   1:  PR[91,2] = PR[90,2] + -28.387;
   1:  PR[91,3] = PR[90,3] + 93.038;
   1:L PR[91] R[100]mm/sec CNT100;
   1:  PR[91,1] = PR[90,1] + 46.902;
   1:  PR[91,2] = PR[90,2] + -26.054;
   1:  PR[91,3] = PR[90,3] + 93.061;
   1:L PR[91] R[100]mm/sec CNT100;
   1:  PR[91,1] = PR[90,1] + 49.030;
   1:  PR[91,2] = PR[90,2] + -24.431;
   1:  PR[91,3] = PR[90,3] + 93.084;
   1:L PR[91] R[100]mm/sec CNT100;
   1:  PR[91,1] = PR[90,1] + 50.984;
   1:  PR[91,2] = PR[90,2] + -22.977;
   1:  PR[91,3] = PR[90,3] + 93.096;
   1:L PR[91] R[100]mm/sec CNT100;
   1:  PR[91,1] = PR[90,1] + 54.397;
   1:  PR[91,2] = PR[90,2] + -19.283;
   1:  PR[91,3] = PR[90,3] + 93.107;
   1:L PR[91] R[100]mm/sec CNT100;
   1:  PR[91,1] = PR[90,1] + 55.453;
   1:  PR[91,2] = PR[90,2] + -17.640;
   1:  PR[91,3] = PR[90,3] + 93.130;
   1:L PR[91] R[100]mm/sec CNT100;
   1:  PR[91,1] = PR[90,1] + 57.214;
   1:  PR[91,2] = PR[90,2] + -15.068;
   1:  PR[91,3] = PR[90,3] + 93.138;
   1:L PR[91] R[100]mm/sec CNT100;
   1:  PR[91,1] = PR[90,1] + 59.274;
   1:  PR[91,2] = PR[90,2] + -10.527;
   1:  PR[91,3] = PR[90,3] + 93.152;
   1:L PR[91] R[100]mm/sec CNT100;
   1:  PR[91,1] = PR[90,1] + 60.517;
   1:  PR[91,2] = PR[90,2] + -5.701;
   1:  PR[91,3] = PR[90,3] + 93.174;
   1:L PR[91] R[100]mm/sec CNT100;
   1:  PR[91,1] = PR[90,1] + 60.793;
   1:  PR[91,2] = PR[90,2] + -2.425;
   1:  PR[91,3] = PR[90,3] + 93.197;
   1:L PR[91] R[100]mm/sec CNT100;
   1:  PR[91,1] = PR[90,1] + 60.883;
   1:  PR[91,2] = PR[90,2] + -0.761;
   1:  PR[91,3] = PR[90,3] + 93.211;
   1:L PR[91] R[100]mm/sec CNT100;
   1:  PR[91,1] = PR[90,1] + 60.748;
   1:  PR[91,2] = PR[90,2] + 0.799;
   1:  PR[91,3] = PR[90,3] + 93.219;
   1:L PR[91] R[100]mm/sec CNT100;
   1:  PR[91,1] = PR[90,1] + 60.667;
   1:  PR[91,2] = PR[90,2] + 2.423;
   1:  PR[91,3] = PR[90,3] + 93.226;
   1:L PR[91] R[100]mm/sec CNT100;
   1:  PR[91,1] = PR[90,1] + 60.517;
   1:  PR[91,2] = PR[90,2] + 4.243;
   1:  PR[91,3] = PR[90,3] + 93.233;
   1:L PR[91] R[100]mm/sec CNT100;
   1:  PR[91,1] = PR[90,1] + 59.274;
   1:  PR[91,2] = PR[90,2] + 9.068;
   1:  PR[91,3] = PR[90,3] + 93.241;
   1:L PR[91] R[100]mm/sec CNT100;
   1:  PR[91,1] = PR[90,1] + 57.214;
   1:  PR[91,2] = PR[90,2] + 13.609;
   1:  PR[91,3] = PR[90,3] + 93.263;
   1:L PR[91] R[100]mm/sec CNT100;
   1:  PR[91,1] = PR[90,1] + 55.453;
   1:  PR[91,2] = PR[90,2] + 16.181;
   1:  PR[91,3] = PR[90,3] + 93.285;
   1:L PR[91] R[100]mm/sec CNT100;
   1:  PR[91,1] = PR[90,1] + 54.397;
   1:  PR[91,2] = PR[90,2] + 17.825;
   1:  PR[91,3] = PR[90,3] + 93.299;
   1:L PR[91] R[100]mm/sec CNT100;
   1:  PR[91,1] = PR[90,1] + 50.984;
   1:  PR[91,2] = PR[90,2] + 21.518;
   1:  PR[91,3] = PR[90,3] + 93.308;
   1:L PR[91] R[100]mm/sec CNT100;
   1:  PR[91,1] = PR[90,1] + 49.030;
   1:  PR[91,2] = PR[90,2] + 22.972;
   1:  PR[91,3] = PR[90,3] + 93.330;
   1:L PR[91] R[100]mm/sec CNT100;
   1:  PR[91,1] = PR[90,1] + 46.902;
   1:  PR[91,2] = PR[90,2] + 24.595;
   1:  PR[91,3] = PR[90,3] + 93.341;
   1:L PR[91] R[100]mm/sec CNT100;
   1:  PR[91,1] = PR[90,1] + 42.292;
   1:  PR[91,2] = PR[90,2] + 26.928;
   1:  PR[91,3] = PR[90,3] + 93.353;
   1:L PR[91] R[100]mm/sec CNT100;
   1:  PR[91,1] = PR[90,1] + 37.245;
   1:  PR[91,2] = PR[90,2] + 28.447;
   1:  PR[91,3] = PR[90,3] + 93.376;
   1:L PR[91] R[100]mm/sec CNT100;
   1:  PR[91,1] = PR[90,1] + 32.511;
   1:  PR[91,2] = PR[90,2] + 29.043;
   1:  PR[91,3] = PR[90,3] + 93.399;
   1:L PR[91] R[100]mm/sec CNT100;
   1:  PR[91,1] = PR[90,1] + 31.765;
   1:  PR[91,2] = PR[90,2] + 29.058;
   1:  PR[91,3] = PR[90,3] + 93.421;
   1:L PR[91] R[100]mm/sec CNT100;
   1:  PR[91,1] = PR[90,1] + 27.568;
   1:  PR[91,2] = PR[90,2] + 28.827;
   1:  PR[91,3] = PR[90,3] + 93.424;
   1:L PR[91] R[100]mm/sec CNT100;
   1:  PR[91,1] = PR[90,1] + 26.159;
   1:  PR[91,2] = PR[90,2] + 28.598;
   1:  PR[91,3] = PR[90,3] + 93.443;
   1:L PR[91] R[100]mm/sec CNT100;
   1:  PR[91,1] = PR[90,1] + 21.407;
   1:  PR[91,2] = PR[90,2] + 27.464;
   1:  PR[91,3] = PR[90,3] + 93.449;
   1:L PR[91] R[100]mm/sec CNT100;
   1:  PR[91,1] = PR[90,1] + 20.575;
   1:  PR[91,2] = PR[90,2] + 27.472;
   1:  PR[91,3] = PR[90,3] + 93.471;
   1:L PR[91] R[100]mm/sec CNT100;
   1:  PR[91,1] = PR[90,1] + 19.235;
   1:  PR[91,2] = PR[90,2] + 27.410;
   1:  PR[91,3] = PR[90,3] + 93.474;
   1:L PR[91] R[100]mm/sec CNT100;
   1:  PR[91,1] = PR[90,1] + 18.275;
   1:  PR[91,2] = PR[90,2] + 27.467;
   1:  PR[91,3] = PR[90,3] + 93.480;
   1:L PR[91] R[100]mm/sec CNT100;
   1:  PR[91,1] = PR[90,1] + 7.525;
   1:  PR[91,2] = PR[90,2] + 27.884;
   1:  PR[91,3] = PR[90,3] + 93.485;
   1:L PR[91] R[100]mm/sec CNT100;
   1:  PR[91,1] = PR[90,1] + -2.993;
   1:  PR[91,2] = PR[90,2] + 27.478;
   1:  PR[91,3] = PR[90,3] + 93.533;
   1:L PR[91] R[100]mm/sec CNT100;
   1:  PR[91,1] = PR[90,1] + -5.796;
   1:  PR[91,2] = PR[90,2] + 27.186;
   1:  PR[91,3] = PR[90,3] + 93.579;
   1:L PR[91] R[100]mm/sec CNT100;
   1:  PR[91,1] = PR[90,1] + -13.027;
   1:  PR[91,2] = PR[90,2] + 26.396;
   1:  PR[91,3] = PR[90,3] + 93.592;
   1:L PR[91] R[100]mm/sec CNT100;
   1:  PR[91,1] = PR[90,1] + -18.279;
   1:  PR[91,2] = PR[90,2] + 25.461;
   1:  PR[91,3] = PR[90,3] + 93.624;
   1:L PR[91] R[100]mm/sec CNT100;
   1:  PR[91,1] = PR[90,1] + -22.384;
   1:  PR[91,2] = PR[90,2] + 24.710;
   1:  PR[91,3] = PR[90,3] + 93.648;
   1:L PR[91] R[100]mm/sec CNT100;
   1:  PR[91,1] = PR[90,1] + -30.899;
   1:  PR[91,2] = PR[90,2] + 22.489;
   1:  PR[91,3] = PR[90,3] + 93.667;
   1:L PR[91] R[100]mm/sec CNT100;
   1:  PR[91,1] = PR[90,1] + -36.804;
   1:  PR[91,2] = PR[90,2] + 20.391;
   1:  PR[91,3] = PR[90,3] + 93.706;
   1:L PR[91] R[100]mm/sec CNT100;
   1:  PR[91,1] = PR[90,1] + -37.835;
   1:  PR[91,2] = PR[90,2] + 19.997;
   1:  PR[91,3] = PR[90,3] + 93.734;
   1:L PR[91] R[100]mm/sec CNT100;
   1:  PR[91,1] = PR[90,1] + -38.951;
   1:  PR[91,2] = PR[90,2] + 19.482;
   1:  PR[91,3] = PR[90,3] + 93.739;
   1:L PR[91] R[100]mm/sec CNT100;
   1:  PR[91,1] = PR[90,1] + -43.041;
   1:  PR[91,2] = PR[90,2] + 17.397;
   1:  PR[91,3] = PR[90,3] + 93.744;
   1:L PR[91] R[100]mm/sec CNT100;
   1:  PR[91,1] = PR[90,1] + -48.727;
   1:  PR[91,2] = PR[90,2] + 13.596;
   1:  PR[91,3] = PR[90,3] + 93.765;
   1:L PR[91] R[100]mm/sec CNT100;
   1:  PR[91] = PR[90];
   1:  PR[91,1] = PR[90,1] + -49.365;
   1:  PR[91,2] = PR[90,2] + 11.172;
   1:  PR[91,3] = PR[90,3] + 95.095;
   1:L PR[91] R[100]mm/sec CNT100;
   1:  PR[91,1] = PR[90,1] + -51.153;
   1:  PR[91,2] = PR[90,2] + 9.107;
   1:  PR[91,3] = PR[90,3] + 93.811;
   1:L PR[91] R[100]mm/sec CNT100;
   1:  PR[91,1] = PR[90,1] + -51.534;
   1:  PR[91,2] = PR[90,2] + 8.367;
   1:  PR[91,3] = PR[90,3] + 93.823;
   1:L PR[91] R[100]mm/sec CNT100;
   1:  PR[91,1] = PR[90,1] + -53.546;
   1:  PR[91,2] = PR[90,2] + 4.268;
   1:  PR[91,3] = PR[90,3] + 93.827;
   1:L PR[91] R[100]mm/sec CNT100;
   1:  PR[91,1] = PR[90,1] + -53.848;
   1:  PR[91,2] = PR[90,2] + 2.477;
   1:  PR[91,3] = PR[90,3] + 93.847;
   1:L PR[91] R[100]mm/sec CNT100;
   1:  PR[91,1] = PR[90,1] + -54.520;
   1:  PR[91,2] = PR[90,2] + -0.745;
   1:  PR[91,3] = PR[90,3] + 93.856;
   1:L PR[91] R[100]mm/sec CNT100;
   1:  PR[91,1] = PR[90,1] + -54.513;
   1:  PR[91,2] = PR[90,2] + -0.783;
   1:  PR[91,3] = PR[90,3] + 93.870;
   1:L PR[91] R[100]mm/sec CNT100;
   1:  PR[91,1] = PR[90,1] + -54.240;
   1:  PR[91,2] = PR[90,2] + -1.528;
   1:  PR[91,3] = PR[90,3] + 93.871;
   1:L PR[91] R[100]mm/sec CNT100;
   1:  PR[91,1] = PR[90,1] + -53.592;
   1:  PR[91,2] = PR[90,2] + -5.660;
   1:  PR[91,3] = PR[90,3] + 93.874;
   1:L PR[91] R[100]mm/sec CNT100;
   1:  PR[91,1] = PR[90,1] + -53.290;
   1:  PR[91,2] = PR[90,2] + -6.306;
   1:  PR[91,3] = PR[90,3] + 93.893;
   1:L PR[91] R[100]mm/sec CNT100;
   1:  PR[91,1] = PR[90,1] + -51.237;
   1:  PR[91,2] = PR[90,2] + -10.564;
   1:  PR[91,3] = PR[90,3] + 93.896;
   1:L PR[91] R[100]mm/sec CNT100;
   1:  PR[91,1] = PR[90,1] + -50.866;
   1:  PR[91,2] = PR[90,2] + -11.004;
   1:  PR[91,3] = PR[90,3] + 93.917;
   1:L PR[91] R[100]mm/sec CNT100;
   1:  PR[91,1] = PR[90,1] + -47.495;
   1:  PR[91,2] = PR[90,2] + -14.421;
   1:  PR[91,3] = PR[90,3] + 93.920;
   1:L PR[91] R[100]mm/sec CNT100;
   1:  PR[91,1] = PR[90,1] + -46.719;
   1:  PR[91,2] = PR[90,2] + -15.165;
   1:  PR[91,3] = PR[90,3] + 93.942;
   1:L PR[91] R[100]mm/sec CNT100;
   1:  PR[91,1] = PR[90,1] + -44.576;
   1:  PR[91,2] = PR[90,2] + -16.660;
   1:  PR[91,3] = PR[90,3] + 93.946;
   1:L PR[91] R[100]mm/sec CNT100;
   1:  PR[91,1] = PR[90,1] + -41.398;
   1:  PR[91,2] = PR[90,2] + -18.787;
   1:  PR[91,3] = PR[90,3] + 93.958;
   1:L PR[91] R[100]mm/sec CNT100;
   1:  PR[91,1] = PR[90,1] + -37.258;
   1:  PR[91,2] = PR[90,2] + -20.921;
   1:  PR[91,3] = PR[90,3] + 93.975;
   1:L PR[91] R[100]mm/sec CNT100;
   1:  PR[91,1] = PR[90,1] + -36.150;
   1:  PR[91,2] = PR[90,2] + -21.445;
   1:  PR[91,3] = PR[90,3] + 93.996;
   1:L PR[91] R[100]mm/sec CNT100;
   1:  PR[91,1] = PR[90,1] + -28.560;
   1:  PR[91,2] = PR[90,2] + -24.144;
   1:  PR[91,3] = PR[90,3] + 94.002;
   1:L PR[91] R[100]mm/sec CNT100;
   1:  PR[91,1] = PR[90,1] + -19.983;
   1:  PR[91,2] = PR[90,2] + -26.385;
   1:  PR[91,3] = PR[90,3] + 94.038;
   1:L PR[91] R[100]mm/sec CNT100;
   1:  PR[91,1] = PR[90,1] + -15.009;
   1:  PR[91,2] = PR[90,2] + -27.294;
   1:  PR[91,3] = PR[90,3] + 94.078;
   1:L PR[91] R[100]mm/sec CNT100;
   1:  PR[91,1] = PR[90,1] + -10.557;
   1:  PR[91,2] = PR[90,2] + -28.087;
   1:  PR[91,3] = PR[90,3] + 94.101;
   1:L PR[91] R[100]mm/sec CNT100;
   1:  PR[91,1] = PR[90,1] + -0.444;
   1:  PR[91,2] = PR[90,2] + -29.181;
   1:  PR[91,3] = PR[90,3] + 94.121;
   1:L PR[91] R[100]mm/sec CNT100;
   1:  PR[91,1] = PR[90,1] + 6.896;
   1:  PR[91,2] = PR[90,2] + -29.464;
   1:  PR[91,3] = PR[90,3] + 94.167;
   1:L PR[91] R[100]mm/sec CNT100;
   1:  PR[91,1] = PR[90,1] + 9.665;
   1:  PR[91,2] = PR[90,2] + -29.600;
   1:  PR[91,3] = PR[90,3] + 94.200;
   1:L PR[91] R[100]mm/sec CNT100;
   1:  PR[91,1] = PR[90,1] + 13.880;
   1:  PR[91,2] = PR[90,2] + -29.451;
   1:  PR[91,3] = PR[90,3] + 94.212;
   1:L PR[91] R[100]mm/sec CNT100;
   1:  PR[91,1] = PR[90,1] + 21.353;
   1:  PR[91,2] = PR[90,2] + -29.130;
   1:  PR[91,3] = PR[90,3] + 94.231;
   1:L PR[91] R[100]mm/sec CNT100;
   1:  PR[91,1] = PR[90,1] + 25.563;
   1:  PR[91,2] = PR[90,2] + -30.127;
   1:  PR[91,3] = PR[90,3] + 94.265;
   1:L PR[91] R[100]mm/sec CNT100;
   1:  PR[91,1] = PR[90,1] + 27.869;
   1:  PR[91,2] = PR[90,2] + -30.501;
   1:  PR[91,3] = PR[90,3] + 94.284;
   1:L PR[91] R[100]mm/sec CNT100;
   1:  PR[91,1] = PR[90,1] + 31.160;
   1:  PR[91,2] = PR[90,2] + -30.682;
   1:  PR[91,3] = PR[90,3] + 94.295;
   1:L PR[91] R[100]mm/sec CNT100;
   1:  PR[91,1] = PR[90,1] + 32.947;
   1:  PR[91,2] = PR[90,2] + -30.648;
   1:  PR[91,3] = PR[90,3] + 94.310;
   1:L PR[91] R[100]mm/sec CNT100;
   1:  PR[91,1] = PR[90,1] + 36.769;
   1:  PR[91,2] = PR[90,2] + -30.166;
   1:  PR[91,3] = PR[90,3] + 94.318;
   1:L PR[91] R[100]mm/sec CNT100;
   1:  PR[91,1] = PR[90,1] + 37.799;
   1:  PR[91,2] = PR[90,2] + -29.954;
   1:  PR[91,3] = PR[90,3] + 94.335;
   1:L PR[91] R[100]mm/sec CNT100;
   1:  PR[91,1] = PR[90,1] + 42.128;
   1:  PR[91,2] = PR[90,2] + -28.597;
   1:  PR[91,3] = PR[90,3] + 94.340;
   1:L PR[91] R[100]mm/sec CNT100;
   1:  PR[91,1] = PR[90,1] + 42.265;
   1:  PR[91,2] = PR[90,2] + -28.541;
   1:  PR[91,3] = PR[90,3] + 94.360;
   1:L PR[91] R[100]mm/sec CNT100;
   1:  PR[91,1] = PR[90,1] + 43.627;
   1:  PR[91,2] = PR[90,2] + -27.829;
   1:  PR[91,3] = PR[90,3] + 94.361;
   1:L PR[91] R[100]mm/sec CNT100;
   1:  PR[91,1] = PR[90,1] + 46.813;
   1:  PR[91,2] = PR[90,2] + -26.224;
   1:  PR[91,3] = PR[90,3] + 94.368;
   1:L PR[91] R[100]mm/sec CNT100;
   1:  PR[91,1] = PR[90,1] + 50.933;
   1:  PR[91,2] = PR[90,2] + -23.145;
   1:  PR[91,3] = PR[90,3] + 94.384;
   1:L PR[91] R[100]mm/sec CNT100;
   1:  PR[91,1] = PR[90,1] + 52.529;
   1:  PR[91,2] = PR[90,2] + -21.411;
   1:  PR[91,3] = PR[90,3] + 94.407;
   1:L PR[91] R[100]mm/sec CNT100;
   1:  PR[91,1] = PR[90,1] + 54.411;
   1:  PR[91,2] = PR[90,2] + -19.423;
   1:  PR[91,3] = PR[90,3] + 94.418;
   1:L PR[91] R[100]mm/sec CNT100;
   1:  PR[91,1] = PR[90,1] + 56.574;
   1:  PR[91,2] = PR[90,2] + -16.056;
   1:  PR[91,3] = PR[90,3] + 94.430;
   1:L PR[91] R[100]mm/sec CNT100;
   1:  PR[91,1] = PR[90,1] + 57.151;
   1:  PR[91,2] = PR[90,2] + -15.186;
   1:  PR[91,3] = PR[90,3] + 94.448;
   1:L PR[91] R[100]mm/sec CNT100;
   1:  PR[91,1] = PR[90,1] + 58.813;
   1:  PR[91,2] = PR[90,2] + -11.280;
   1:  PR[91,3] = PR[90,3] + 94.453;
   1:L PR[91] R[100]mm/sec CNT100;
   1:  PR[91,1] = PR[90,1] + 59.145;
   1:  PR[91,2] = PR[90,2] + -10.551;
   1:  PR[91,3] = PR[90,3] + 94.472;
   1:L PR[91] R[100]mm/sec CNT100;
   1:  PR[91,1] = PR[90,1] + 60.403;
   1:  PR[91,2] = PR[90,2] + -5.711;
   1:  PR[91,3] = PR[90,3] + 94.475;
   1:L PR[91] R[100]mm/sec CNT100;
   1:  PR[91,1] = PR[90,1] + 60.481;
   1:  PR[91,2] = PR[90,2] + -4.788;
   1:  PR[91,3] = PR[90,3] + 94.498;
   1:L PR[91] R[100]mm/sec CNT100;
   1:  PR[91,1] = PR[90,1] + 60.550;
   1:  PR[91,2] = PR[90,2] + -3.505;
   1:  PR[91,3] = PR[90,3] + 94.502;
   1:L PR[91] R[100]mm/sec CNT100;
   1:  PR[91,1] = PR[90,1] + 60.782;
   1:  PR[91,2] = PR[90,2] + -0.697;
   1:  PR[91,3] = PR[90,3] + 94.508;
   1:L PR[91] R[100]mm/sec CNT100;
   1:  PR[91,1] = PR[90,1] + 60.735;
   1:  PR[91,2] = PR[90,2] + 0.247;
   1:  PR[91,3] = PR[90,3] + 94.521;
   1:L PR[91] R[100]mm/sec CNT100;
   1:  PR[91,1] = PR[90,1] + 60.403;
   1:  PR[91,2] = PR[90,2] + 4.253;
   1:  PR[91,3] = PR[90,3] + 94.525;
   1:L PR[91] R[100]mm/sec CNT100;
   1:  PR[91,1] = PR[90,1] + 59.145;
   1:  PR[91,2] = PR[90,2] + 9.092;
   1:  PR[91,3] = PR[90,3] + 94.543;
   1:L PR[91] R[100]mm/sec CNT100;
   1:  PR[91,1] = PR[90,1] + 58.813;
   1:  PR[91,2] = PR[90,2] + 9.821;
   1:  PR[91,3] = PR[90,3] + 94.565;
   1:L PR[91] R[100]mm/sec CNT100;
   1:  PR[91,1] = PR[90,1] + 57.151;
   1:  PR[91,2] = PR[90,2] + 13.728;
   1:  PR[91,3] = PR[90,3] + 94.569;
   1:L PR[91] R[100]mm/sec CNT100;
   1:  PR[91,1] = PR[90,1] + 56.574;
   1:  PR[91,2] = PR[90,2] + 14.597;
   1:  PR[91,3] = PR[90,3] + 94.588;
   1:L PR[91] R[100]mm/sec CNT100;
   1:  PR[91,1] = PR[90,1] + 54.411;
   1:  PR[91,2] = PR[90,2] + 17.964;
   1:  PR[91,3] = PR[90,3] + 94.593;
   1:L PR[91] R[100]mm/sec CNT100;
   1:  PR[91,1] = PR[90,1] + 52.529;
   1:  PR[91,2] = PR[90,2] + 19.953;
   1:  PR[91,3] = PR[90,3] + 94.611;
   1:L PR[91] R[100]mm/sec CNT100;
   1:  PR[91,1] = PR[90,1] + 50.933;
   1:  PR[91,2] = PR[90,2] + 21.686;
   1:  PR[91,3] = PR[90,3] + 94.623;
   1:L PR[91] R[100]mm/sec CNT100;
   1:  PR[91,1] = PR[90,1] + 46.813;
   1:  PR[91,2] = PR[90,2] + 24.766;
   1:  PR[91,3] = PR[90,3] + 94.634;
   1:L PR[91] R[100]mm/sec CNT100;
   1:  PR[91,1] = PR[90,1] + 43.627;
   1:  PR[91,2] = PR[90,2] + 26.370;
   1:  PR[91,3] = PR[90,3] + 94.657;
   1:L PR[91] R[100]mm/sec CNT100;
   1:  PR[91,1] = PR[90,1] + 42.266;
   1:  PR[91,2] = PR[90,2] + 27.082;
   1:  PR[91,3] = PR[90,3] + 94.673;
   1:L PR[91] R[100]mm/sec CNT100;
   1:  PR[91,1] = PR[90,1] + 42.128;
   1:  PR[91,2] = PR[90,2] + 27.139;
   1:  PR[91,3] = PR[90,3] + 94.680;
   1:L PR[91] R[100]mm/sec CNT100;
   1:  PR[91,1] = PR[90,1] + 37.800;
   1:  PR[91,2] = PR[90,2] + 28.494;
   1:L PR[91] R[100]mm/sec CNT100;
   1:  PR[91,1] = PR[90,1] + 36.772;
   1:  PR[91,2] = PR[90,2] + 28.707;
   1:  PR[91,3] = PR[90,3] + 94.701;
   1:L PR[91] R[100]mm/sec CNT100;
   1:  PR[91,1] = PR[90,1] + 32.950;
   1:  PR[91,2] = PR[90,2] + 29.189;
   1:  PR[91,3] = PR[90,3] + 94.706;
   1:L PR[91] R[100]mm/sec CNT100;
   1:  PR[91,1] = PR[90,1] + 31.164;
   1:  PR[91,2] = PR[90,2] + 29.224;
   1:  PR[91,3] = PR[90,3] + 94.723;
   1:L PR[91] R[100]mm/sec CNT100;
   1:  PR[91,1] = PR[90,1] + 27.875;
   1:  PR[91,2] = PR[90,2] + 29.043;
   1:  PR[91,3] = PR[90,3] + 94.731;
   1:L PR[91] R[100]mm/sec CNT100;
   1:  PR[91,1] = PR[90,1] + 25.550;
   1:  PR[91,2] = PR[90,2] + 28.666;
   1:  PR[91,3] = PR[90,3] + 94.746;
   1:L PR[91] R[100]mm/sec CNT100;
   1:  PR[91,1] = PR[90,1] + 21.358;
   1:  PR[91,2] = PR[90,2] + 27.673;
   1:  PR[91,3] = PR[90,3] + 94.756;
   1:L PR[91] R[100]mm/sec CNT100;
   1:  PR[91,1] = PR[90,1] + 9.661;
   1:  PR[91,2] = PR[90,2] + 28.141;
   1:  PR[91,3] = PR[90,3] + 94.776;
   1:L PR[91] R[100]mm/sec CNT100;
   1:  PR[91,1] = PR[90,1] + 6.896;
   1:  PR[91,2] = PR[90,2] + 28.005;
   1:  PR[91,3] = PR[90,3] + 94.828;
   1:L PR[91] R[100]mm/sec CNT100;
   1:  PR[91,1] = PR[90,1] + -0.444;
   1:  PR[91,2] = PR[90,2] + 27.723;
   1:  PR[91,3] = PR[90,3] + 94.841;
   1:L PR[91] R[100]mm/sec CNT100;
   1:  PR[91,1] = PR[90,1] + -10.557;
   1:  PR[91,2] = PR[90,2] + 26.628;
   1:  PR[91,3] = PR[90,3] + 94.874;
   1:L PR[91] R[100]mm/sec CNT100;
   1:  PR[91,1] = PR[90,1] + -15.009;
   1:  PR[91,2] = PR[90,2] + 25.835;
   1:  PR[91,3] = PR[90,3] + 94.920;
   1:L PR[91] R[100]mm/sec CNT100;
   1:  PR[91,1] = PR[90,1] + -19.983;
   1:  PR[91,2] = PR[90,2] + 24.926;
   1:  PR[91,3] = PR[90,3] + 94.940;
   1:L PR[91] R[100]mm/sec CNT100;
   1:  PR[91,1] = PR[90,1] + -28.560;
   1:  PR[91,2] = PR[90,2] + 22.685;
   1:  PR[91,3] = PR[90,3] + 94.963;
   1:L PR[91] R[100]mm/sec CNT100;
   1:  PR[91,1] = PR[90,1] + -36.150;
   1:  PR[91,2] = PR[90,2] + 19.987;
   1:  PR[91,3] = PR[90,3] + 95.003;
   1:L PR[91] R[100]mm/sec CNT100;
   1:  PR[91,1] = PR[90,1] + -37.263;
   1:  PR[91,2] = PR[90,2] + 19.461;
   1:  PR[91,3] = PR[90,3] + 95.039;
   1:L PR[91] R[100]mm/sec CNT100;
   1:  PR[91,1] = PR[90,1] + -41.425;
   1:  PR[91,2] = PR[90,2] + 17.338;
   1:  PR[91,3] = PR[90,3] + 95.044;
   1:L PR[91] R[100]mm/sec CNT100;
   1:  PR[91,1] = PR[90,1] + -45.308;
   1:  PR[91,2] = PR[90,2] + 14.742;
   1:  PR[91,3] = PR[90,3] + 95.065;
   1:L PR[91] R[100]mm/sec CNT100;
   1:  PR[91,1] = PR[90,1] + -46.871;
   1:  PR[91,2] = PR[90,2] + 13.661;
   1:  PR[91,3] = PR[90,3] + 95.086;
   1:L PR[91] R[100]mm/sec CNT100;
   1:  PR[91] = PR[90];
   1:  PR[91,1] = PR[90,1] + -49.712;
   1:  PR[91,2] = PR[90,2] + 9.014;
   1:  PR[91,3] = PR[90,3] + 96.395;
   1:L PR[91] R[100]mm/sec CNT100;
   1:  PR[91,1] = PR[90,1] + -49.895;
   1:  PR[91,2] = PR[90,2] + 8.687;
   1:  PR[91,3] = PR[90,3] + 95.126;
   1:L PR[91] R[100]mm/sec CNT100;
   1:  PR[91,1] = PR[90,1] + -52.067;
   1:  PR[91,2] = PR[90,2] + 4.259;
   1:  PR[91,3] = PR[90,3] + 95.127;
   1:L PR[91] R[100]mm/sec CNT100;
   1:  PR[91,1] = PR[90,1] + -52.198;
   1:  PR[91,2] = PR[90,2] + 3.486;
   1:  PR[91,3] = PR[90,3] + 95.150;
   1:L PR[91] R[100]mm/sec CNT100;
   1:  PR[91,1] = PR[90,1] + -52.873;
   1:  PR[91,2] = PR[90,2] + 0.250;
   1:  PR[91,3] = PR[90,3] + 95.153;
   1:L PR[91] R[100]mm/sec CNT100;
   1:  PR[91,1] = PR[90,1] + -53.010;
   1:  PR[91,2] = PR[90,2] + -0.543;
   1:  PR[91,3] = PR[90,3] + 95.168;
   1:L PR[91] R[100]mm/sec CNT100;
   1:  PR[91,1] = PR[90,1] + -52.918;
   1:  PR[91,2] = PR[90,2] + -0.793;
   1:  PR[91,3] = PR[90,3] + 95.172;
   1:L PR[91] R[100]mm/sec CNT100;
   1:  PR[91,1] = PR[90,1] + -52.146;
   1:  PR[91,2] = PR[90,2] + -5.720;
   1:  PR[91,3] = PR[90,3] + 95.173;
   1:L PR[91] R[100]mm/sec CNT100;
   1:  PR[91,1] = PR[90,1] + -51.429;
   1:  PR[91,2] = PR[90,2] + -7.208;
   1:  PR[91,3] = PR[90,3] + 95.196;
   1:L PR[91] R[100]mm/sec CNT100;
   1:  PR[91,1] = PR[90,1] + -49.680;
   1:  PR[91,2] = PR[90,2] + -10.338;
   1:  PR[91,3] = PR[90,3] + 95.203;
   1:L PR[91] R[100]mm/sec CNT100;
   1:  PR[91,1] = PR[90,1] + -49.463;
   1:  PR[91,2] = PR[90,2] + -10.639;
   1:  PR[91,3] = PR[90,3] + 95.219;
   1:L PR[91] R[100]mm/sec CNT100;
   1:  PR[91,1] = PR[90,1] + -46.177;
   1:  PR[91,2] = PR[90,2] + -13.970;
   1:  PR[91,3] = PR[90,3] + 95.221;
   1:L PR[91] R[100]mm/sec CNT100;
   1:  PR[91,1] = PR[90,1] + -44.827;
   1:  PR[91,2] = PR[90,2] + -15.265;
   1:  PR[91,3] = PR[90,3] + 95.242;
   1:L PR[91] R[100]mm/sec CNT100;
   1:  PR[91,1] = PR[90,1] + -41.238;
   1:  PR[91,2] = PR[90,2] + -17.768;
   1:  PR[91,3] = PR[90,3] + 95.251;
   1:L PR[91] R[100]mm/sec CNT100;
   1:  PR[91,1] = PR[90,1] + -39.794;
   1:  PR[91,2] = PR[90,2] + -18.734;
   1:  PR[91,3] = PR[90,3] + 95.270;
   1:L PR[91] R[100]mm/sec CNT100;
   1:  PR[91,1] = PR[90,1] + -37.907;
   1:  PR[91,2] = PR[90,2] + -19.708;
   1:  PR[91,3] = PR[90,3] + 95.278;
   1:L PR[91] R[100]mm/sec CNT100;
   1:  PR[91,1] = PR[90,1] + -33.865;
   1:  PR[91,2] = PR[90,2] + -21.618;
   1:  PR[91,3] = PR[90,3] + 95.288;
   1:L PR[91] R[100]mm/sec CNT100;
   1:  PR[91,1] = PR[90,1] + -26.220;
   1:  PR[91,2] = PR[90,2] + -24.340;
   1:  PR[91,3] = PR[90,3] + 95.308;
   1:L PR[91] R[100]mm/sec CNT100;
   1:  PR[91,1] = PR[90,1] + -17.581;
   1:  PR[91,2] = PR[90,2] + -26.600;
   1:  PR[91,3] = PR[90,3] + 95.345;
   1:L PR[91] R[100]mm/sec CNT100;
   1:  PR[91,1] = PR[90,1] + -11.739;
   1:  PR[91,2] = PR[90,2] + -27.669;
   1:  PR[91,3] = PR[90,3] + 95.385;
   1:L PR[91] R[100]mm/sec CNT100;
   1:  PR[91,1] = PR[90,1] + -8.086;
   1:  PR[91,2] = PR[90,2] + -28.319;
   1:  PR[91,3] = PR[90,3] + 95.412;
   1:L PR[91] R[100]mm/sec CNT100;
   1:  PR[91,1] = PR[90,1] + 1.029;
   1:  PR[91,2] = PR[90,2] + -29.314;
   1:  PR[91,3] = PR[90,3] + 95.429;
   1:L PR[91] R[100]mm/sec CNT100;
   1:  PR[91,1] = PR[90,1] + 2.098;
   1:  PR[91,2] = PR[90,2] + -29.426;
   1:  PR[91,3] = PR[90,3] + 95.471;
   1:L PR[91] R[100]mm/sec CNT100;
   1:  PR[91,1] = PR[90,1] + 6.247;
   1:  PR[91,2] = PR[90,2] + -29.586;
   1:  PR[91,3] = PR[90,3] + 95.475;
   1:L PR[91] R[100]mm/sec CNT100;
   1:  PR[91,1] = PR[90,1] + 11.792;
   1:  PR[91,2] = PR[90,2] + -29.857;
   1:  PR[91,3] = PR[90,3] + 95.494;
   1:L PR[91] R[100]mm/sec CNT100;
   1:  PR[91,1] = PR[90,1] + 14.899;
   1:  PR[91,2] = PR[90,2] + -29.747;
   1:  PR[91,3] = PR[90,3] + 95.519;
   1:L PR[91] R[100]mm/sec CNT100;
   1:  PR[91,1] = PR[90,1] + 20.303;
   1:  PR[91,2] = PR[90,2] + -29.520;
   1:  PR[91,3] = PR[90,3] + 95.533;
   1:L PR[91] R[100]mm/sec CNT100;
   1:  PR[91,1] = PR[90,1] + 24.444;
   1:  PR[91,2] = PR[90,2] + -29.300;
   1:  PR[91,3] = PR[90,3] + 95.558;
   1:L PR[91] R[100]mm/sec CNT100;
   1:  PR[91,1] = PR[90,1] + 24.240;
   1:  PR[91,2] = PR[90,2] + -30.026;
   1:  PR[91,3] = PR[90,3] + 95.577;
   1:L PR[91] R[100]mm/sec CNT100;
   1:  PR[91,1] = PR[90,1] + 24.959;
   1:  PR[91,2] = PR[90,2] + -30.195;
   1:  PR[91,3] = PR[90,3] + 95.580;
   1:L PR[91] R[100]mm/sec CNT100;
   1:  PR[91,1] = PR[90,1] + 28.174;
   1:  PR[91,2] = PR[90,2] + -30.717;
   1:  PR[91,3] = PR[90,3] + 95.583;
   1:L PR[91] R[100]mm/sec CNT100;
   1:  PR[91,1] = PR[90,1] + 30.556;
   1:  PR[91,2] = PR[90,2] + -30.848;
   1:  PR[91,3] = PR[90,3] + 95.598;
   1:L PR[91] R[100]mm/sec CNT100;
   1:  PR[91,1] = PR[90,1] + 33.384;
   1:  PR[91,2] = PR[90,2] + -30.793;
   1:  PR[91,3] = PR[90,3] + 95.609;
   1:L PR[91] R[100]mm/sec CNT100;
   1:  PR[91,1] = PR[90,1] + 36.206;
   1:  PR[91,2] = PR[90,2] + -30.438;
   1:  PR[91,3] = PR[90,3] + 95.622;
   1:L PR[91] R[100]mm/sec CNT100;
   1:  PR[91,1] = PR[90,1] + 38.380;
   1:  PR[91,2] = PR[90,2] + -29.988;
   1:  PR[91,3] = PR[90,3] + 95.635;
   1:L PR[91] R[100]mm/sec CNT100;
   1:  PR[91,1] = PR[90,1] + 41.632;
   1:  PR[91,2] = PR[90,2] + -28.969;
   1:  PR[91,3] = PR[90,3] + 95.645;
   1:L PR[91] R[100]mm/sec CNT100;
   1:  PR[91,1] = PR[90,1] + 42.997;
   1:  PR[91,2] = PR[90,2] + -28.411;
   1:  PR[91,3] = PR[90,3] + 95.660;
   1:L PR[91] R[100]mm/sec CNT100;
   1:  PR[91,1] = PR[90,1] + 46.615;
   1:  PR[91,2] = PR[90,2] + -26.519;
   1:  PR[91,3] = PR[90,3] + 95.667;
   1:L PR[91] R[100]mm/sec CNT100;
   1:  PR[91,1] = PR[90,1] + 47.102;
   1:  PR[91,2] = PR[90,2] + -26.205;
   1:  PR[91,3] = PR[90,3] + 95.685;
   1:L PR[91] R[100]mm/sec CNT100;
   1:  PR[91,1] = PR[90,1] + 49.866;
   1:  PR[91,2] = PR[90,2] + -24.067;
   1:  PR[91,3] = PR[90,3] + 95.688;
   1:L PR[91] R[100]mm/sec CNT100;
   1:  PR[91,1] = PR[90,1] + 50.896;
   1:  PR[91,2] = PR[90,2] + -23.301;
   1:  PR[91,3] = PR[90,3] + 95.704;
   1:L PR[91] R[100]mm/sec CNT100;
   1:  PR[91,1] = PR[90,1] + 54.418;
   1:  PR[91,2] = PR[90,2] + -19.573;
   1:  PR[91,3] = PR[90,3] + 95.710;
   1:L PR[91] R[100]mm/sec CNT100;
   1:  PR[91,1] = PR[90,1] + 55.294;
   1:  PR[91,2] = PR[90,2] + -18.209;
   1:  PR[91,3] = PR[90,3] + 95.733;
   1:L PR[91] R[100]mm/sec CNT100;
   1:  PR[91,1] = PR[90,1] + 57.216;
   1:  PR[91,2] = PR[90,2] + -15.312;
   1:  PR[91,3] = PR[90,3] + 95.740;
   1:L PR[91] R[100]mm/sec CNT100;
   1:  PR[91,1] = PR[90,1] + 58.360;
   1:  PR[91,2] = PR[90,2] + -12.623;
   1:  PR[91,3] = PR[90,3] + 95.756;
   1:L PR[91] R[100]mm/sec CNT100;
   1:  PR[91,1] = PR[90,1] + 59.226;
   1:  PR[91,2] = PR[90,2] + -10.662;
   1:  PR[91,3] = PR[90,3] + 95.769;
   1:L PR[91] R[100]mm/sec CNT100;
   1:  PR[91,1] = PR[90,1] + 60.131;
   1:  PR[91,2] = PR[90,2] + -6.926;
   1:  PR[91,3] = PR[90,3] + 95.779;
   1:L PR[91] R[100]mm/sec CNT100;
   1:  PR[91,1] = PR[90,1] + 60.428;
   1:  PR[91,2] = PR[90,2] + -5.751;
   1:  PR[91,3] = PR[90,3] + 95.796;
   1:L PR[91] R[100]mm/sec CNT100;
   1:  PR[91,1] = PR[90,1] + 60.838;
   1:  PR[91,2] = PR[90,2] + -0.729;
   1:  PR[91,3] = PR[90,3] + 95.802;
   1:L PR[91] R[100]mm/sec CNT100;
   1:  PR[91,1] = PR[90,1] + 60.428;
   1:  PR[91,2] = PR[90,2] + 4.292;
   1:  PR[91,3] = PR[90,3] + 95.825;
   1:L PR[91] R[100]mm/sec CNT100;
   1:  PR[91,1] = PR[90,1] + 60.131;
   1:  PR[91,2] = PR[90,2] + 5.467;
   1:  PR[91,3] = PR[90,3] + 95.847;
   1:L PR[91] R[100]mm/sec CNT100;
   1:  PR[91,1] = PR[90,1] + 59.226;
   1:  PR[91,2] = PR[90,2] + 9.203;
   1:  PR[91,3] = PR[90,3] + 95.853;
   1:L PR[91] R[100]mm/sec CNT100;
   1:  PR[91,1] = PR[90,1] + 58.360;
   1:  PR[91,2] = PR[90,2] + 11.164;
   1:  PR[91,3] = PR[90,3] + 95.870;
   1:L PR[91] R[100]mm/sec CNT100;
   1:  PR[91,1] = PR[90,1] + 57.216;
   1:  PR[91,2] = PR[90,2] + 13.853;
   1:  PR[91,3] = PR[90,3] + 95.880;
   1:L PR[91] R[100]mm/sec CNT100;
   1:  PR[91,1] = PR[90,1] + 55.294;
   1:  PR[91,2] = PR[90,2] + 16.750;
   1:  PR[91,3] = PR[90,3] + 95.893;
   1:L PR[91] R[100]mm/sec CNT100;
   1:  PR[91,1] = PR[90,1] + 54.418;
   1:  PR[91,2] = PR[90,2] + 18.114;
   1:  PR[91,3] = PR[90,3] + 95.909;
   1:L PR[91] R[100]mm/sec CNT100;
   1:  PR[91,1] = PR[90,1] + 50.896;
   1:  PR[91,2] = PR[90,2] + 21.842;
   1:  PR[91,3] = PR[90,3] + 95.916;
   1:L PR[91] R[100]mm/sec CNT100;
   1:  PR[91,1] = PR[90,1] + 49.866;
   1:  PR[91,2] = PR[90,2] + 22.609;
   1:  PR[91,3] = PR[90,3] + 95.940;
   1:L PR[91] R[100]mm/sec CNT100;
   1:  PR[91,1] = PR[90,1] + 47.103;
   1:  PR[91,2] = PR[90,2] + 24.746;
   1:  PR[91,3] = PR[90,3] + 95.945;
   1:L PR[91] R[100]mm/sec CNT100;
   1:  PR[91,1] = PR[90,1] + 46.616;
   1:  PR[91,2] = PR[90,2] + 25.060;
   1:  PR[91,3] = PR[90,3] + 95.961;
   1:L PR[91] R[100]mm/sec CNT100;
   1:  PR[91,1] = PR[90,1] + 42.999;
   1:  PR[91,2] = PR[90,2] + 26.952;
   1:  PR[91,3] = PR[90,3] + 95.964;
   1:L PR[91] R[100]mm/sec CNT100;
   1:  PR[91,1] = PR[90,1] + 41.635;
   1:  PR[91,2] = PR[90,2] + 27.510;
   1:  PR[91,3] = PR[90,3] + 95.982;
   1:L PR[91] R[100]mm/sec CNT100;
   1:  PR[91,1] = PR[90,1] + 38.383;
   1:  PR[91,2] = PR[90,2] + 28.528;
   1:  PR[91,3] = PR[90,3] + 95.989;
   1:L PR[91] R[100]mm/sec CNT100;
   1:  PR[91,1] = PR[90,1] + 36.211;
   1:  PR[91,2] = PR[90,2] + 28.979;
   1:  PR[91,3] = PR[90,3] + 96.004;
   1:L PR[91] R[100]mm/sec CNT100;
   1:  PR[91,1] = PR[90,1] + 33.389;
   1:  PR[91,2] = PR[90,2] + 29.334;
   1:  PR[91,3] = PR[90,3] + 96.014;
   1:L PR[91] R[100]mm/sec CNT100;
   1:  PR[91,1] = PR[90,1] + 30.562;
   1:  PR[91,2] = PR[90,2] + 29.390;
   1:  PR[91,3] = PR[90,3] + 96.027;
   1:L PR[91] R[100]mm/sec CNT100;
   1:  PR[91,1] = PR[90,1] + 28.182;
   1:  PR[91,2] = PR[90,2] + 29.258;
   1:  PR[91,3] = PR[90,3] + 96.040;
   1:L PR[91] R[100]mm/sec CNT100;
   1:  PR[91,1] = PR[90,1] + 24.943;
   1:  PR[91,2] = PR[90,2] + 28.733;
   1:  PR[91,3] = PR[90,3] + 96.051;
   1:L PR[91] R[100]mm/sec CNT100;
   1:  PR[91,1] = PR[90,1] + 21.966;
   1:  PR[91,2] = PR[90,2] + 28.031;
   1:  PR[91,3] = PR[90,3] + 96.066;
   1:L PR[91] R[100]mm/sec CNT100;
   1:  PR[91,1] = PR[90,1] + 20.333;
   1:  PR[91,2] = PR[90,2] + 28.060;
   1:  PR[91,3] = PR[90,3] + 96.080;
   1:L PR[91] R[100]mm/sec CNT100;
   1:  PR[91,1] = PR[90,1] + 11.788;
   1:  PR[91,2] = PR[90,2] + 28.398;
   1:  PR[91,3] = PR[90,3] + 96.087;
   1:L PR[91] R[100]mm/sec CNT100;
   1:  PR[91,1] = PR[90,1] + 6.247;
   1:  PR[91,2] = PR[90,2] + 28.127;
   1:  PR[91,3] = PR[90,3] + 96.126;
   1:L PR[91] R[100]mm/sec CNT100;
   1:  PR[91,1] = PR[90,1] + 2.103;
   1:  PR[91,2] = PR[90,2] + 27.967;
   1:  PR[91,3] = PR[90,3] + 96.151;
   1:L PR[91] R[100]mm/sec CNT100;
   1:  PR[91,1] = PR[90,1] + -8.086;
   1:  PR[91,2] = PR[90,2] + 26.860;
   1:  PR[91,3] = PR[90,3] + 96.170;
   1:L PR[91] R[100]mm/sec CNT100;
   1:  PR[91,1] = PR[90,1] + -11.739;
   1:  PR[91,2] = PR[90,2] + 26.210;
   1:  PR[91,3] = PR[90,3] + 96.216;
   1:L PR[91] R[100]mm/sec CNT100;
   1:  PR[91,1] = PR[90,1] + -17.583;
   1:  PR[91,2] = PR[90,2] + 25.141;
   1:  PR[91,3] = PR[90,3] + 96.233;
   1:L PR[91] R[100]mm/sec CNT100;
   1:  PR[91,1] = PR[90,1] + -23.182;
   1:  PR[91,2] = PR[90,2] + 23.686;
   1:  PR[91,3] = PR[90,3] + 96.260;
   1:L PR[91] R[100]mm/sec CNT100;
   1:  PR[91,1] = PR[90,1] + -26.217;
   1:  PR[91,2] = PR[90,2] + 22.882;
   1:  PR[91,3] = PR[90,3] + 96.286;
   1:L PR[91] R[100]mm/sec CNT100;
   1:  PR[91,1] = PR[90,1] + -33.865;
   1:  PR[91,2] = PR[90,2] + 20.160;
   1:  PR[91,3] = PR[90,3] + 96.300;
   1:L PR[91] R[100]mm/sec CNT100;
   1:  PR[91,1] = PR[90,1] + -37.911;
   1:  PR[91,2] = PR[90,2] + 18.247;
   1:  PR[91,3] = PR[90,3] + 96.337;
   1:L PR[91] R[100]mm/sec CNT100;
   1:  PR[91,1] = PR[90,1] + -39.809;
   1:  PR[91,2] = PR[90,2] + 17.279;
   1:  PR[91,3] = PR[90,3] + 96.357;
   1:L PR[91] R[100]mm/sec CNT100;
   1:  PR[91,1] = PR[90,1] + -41.586;
   1:  PR[91,2] = PR[90,2] + 16.091;
   1:  PR[91,3] = PR[90,3] + 96.367;
   1:L PR[91] R[100]mm/sec CNT100;
   1:  PR[91,1] = PR[90,1] + -44.936;
   1:  PR[91,2] = PR[90,2] + 13.774;
   1:  PR[91,3] = PR[90,3] + 96.377;
   1:L PR[91] R[100]mm/sec CNT100;
   1:  PR[91] = PR[90];
   1:  PR[91,1] = PR[90,1] + -46.060;
   1:  PR[91,2] = PR[90,2] + 10.834;
   1:  PR[91,3] = PR[90,3] + 97.695;
   1:L PR[91] R[100]mm/sec CNT100;
   1:  PR[91,1] = PR[90,1] + -47.622;
   1:  PR[91,2] = PR[90,2] + 9.323;
   1:  PR[91,3] = PR[90,3] + 96.415;
   1:L PR[91] R[100]mm/sec CNT100;
   1:  PR[91,1] = PR[90,1] + -48.087;
   1:  PR[91,2] = PR[90,2] + 8.684;
   1:  PR[91,3] = PR[90,3] + 96.425;
   1:L PR[91] R[100]mm/sec CNT100;
   1:  PR[91,1] = PR[90,1] + -50.599;
   1:  PR[91,2] = PR[90,2] + 4.195;
   1:  PR[91,3] = PR[90,3] + 96.428;
   1:L PR[91] R[100]mm/sec CNT100;
   1:  PR[91,1] = PR[90,1] + -51.439;
   1:  PR[91,2] = PR[90,2] + -0.728;
   1:  PR[91,3] = PR[90,3] + 96.452;
   1:L PR[91] R[100]mm/sec CNT100;
   1:  PR[91,1] = PR[90,1] + -51.125;
   1:  PR[91,2] = PR[90,2] + -2.557;
   1:  PR[91,3] = PR[90,3] + 96.475;
   1:L PR[91] R[100]mm/sec CNT100;
   1:  PR[91,1] = PR[90,1] + -50.510;
   1:  PR[91,2] = PR[90,2] + -5.430;
   1:  PR[91,3] = PR[90,3] + 96.483;
   1:L PR[91] R[100]mm/sec CNT100;
   1:  PR[91,1] = PR[90,1] + -50.477;
   1:  PR[91,2] = PR[90,2] + -5.674;
   1:  PR[91,3] = PR[90,3] + 96.497;
   1:L PR[91] R[100]mm/sec CNT100;
   1:  PR[91,1] = PR[90,1] + -50.419;
   1:  PR[91,2] = PR[90,2] + -5.812;
   1:  PR[91,3] = PR[90,3] + 96.498;
   1:L PR[91] R[100]mm/sec CNT100;
   1:  PR[91,1] = PR[90,1] + -48.096;
   1:  PR[91,2] = PR[90,2] + -9.970;
   1:L PR[91] R[100]mm/sec CNT100;
   1:  PR[91,1] = PR[90,1] + -47.381;
   1:  PR[91,2] = PR[90,2] + -10.962;
   1:  PR[91,3] = PR[90,3] + 96.520;
   1:L PR[91] R[100]mm/sec CNT100;
   1:  PR[91,1] = PR[90,1] + -44.859;
   1:  PR[91,2] = PR[90,2] + -13.519;
   1:  PR[91,3] = PR[90,3] + 96.526;
   1:L PR[91] R[100]mm/sec CNT100;
   1:  PR[91,1] = PR[90,1] + -42.934;
   1:  PR[91,2] = PR[90,2] + -15.364;
   1:  PR[91,3] = PR[90,3] + 96.542;
   1:L PR[91] R[100]mm/sec CNT100;
   1:  PR[91,1] = PR[90,1] + -38.335;
   1:  PR[91,2] = PR[90,2] + -18.573;
   1:  PR[91,3] = PR[90,3] + 96.554;
   1:L PR[91] R[100]mm/sec CNT100;
   1:  PR[91,1] = PR[90,1] + -38.178;
   1:  PR[91,2] = PR[90,2] + -18.672;
   1:  PR[91,3] = PR[90,3] + 96.580;
   1:L PR[91] R[100]mm/sec CNT100;
   1:  PR[91,1] = PR[90,1] + -31.581;
   1:  PR[91,2] = PR[90,2] + -21.791;
   1:  PR[91,3] = PR[90,3] + 96.581;
   1:L PR[91] R[100]mm/sec CNT100;
   1:  PR[91,1] = PR[90,1] + -23.878;
   1:  PR[91,2] = PR[90,2] + -24.537;
   1:  PR[91,3] = PR[90,3] + 96.614;
   1:L PR[91] R[100]mm/sec CNT100;
   1:  PR[91,1] = PR[90,1] + -20.066;
   1:  PR[91,2] = PR[90,2] + -25.546;
   1:  PR[91,3] = PR[90,3] + 96.652;
   1:L PR[91] R[100]mm/sec CNT100;
   1:  PR[91,1] = PR[90,1] + -15.183;
   1:  PR[91,2] = PR[90,2] + -26.815;
   1:  PR[91,3] = PR[90,3] + 96.670;
   1:L PR[91] R[100]mm/sec CNT100;
   1:  PR[91,1] = PR[90,1] + -5.612;
   1:  PR[91,2] = PR[90,2] + -28.552;
   1:  PR[91,3] = PR[90,3] + 96.693;
   1:L PR[91] R[100]mm/sec CNT100;
   1:  PR[91,1] = PR[90,1] + 4.658;
   1:  PR[91,2] = PR[90,2] + -29.672;
   1:  PR[91,3] = PR[90,3] + 96.737;
   1:L PR[91] R[100]mm/sec CNT100;
   1:  PR[91,1] = PR[90,1] + 13.913;
   1:  PR[91,2] = PR[90,2] + -30.115;
   1:  PR[91,3] = PR[90,3] + 96.785;
   1:L PR[91] R[100]mm/sec CNT100;
   1:  PR[91,1] = PR[90,1] + 19.447;
   1:  PR[91,2] = PR[90,2] + -29.895;
   1:  PR[91,3] = PR[90,3] + 96.827;
   1:L PR[91] R[100]mm/sec CNT100;
   1:  PR[91,1] = PR[90,1] + 25.046;
   1:  PR[91,2] = PR[90,2] + -29.598;
   1:  PR[91,3] = PR[90,3] + 96.852;
   1:L PR[91] R[100]mm/sec CNT100;
   1:  PR[91,1] = PR[90,1] + 24.837;
   1:  PR[91,2] = PR[90,2] + -30.342;
   1:  PR[91,3] = PR[90,3] + 96.878;
   1:L PR[91] R[100]mm/sec CNT100;
   1:  PR[91,1] = PR[90,1] + 28.479;
   1:  PR[91,2] = PR[90,2] + -30.933;
   1:  PR[91,3] = PR[90,3] + 96.881;
   1:L PR[91] R[100]mm/sec CNT100;
   1:  PR[91,1] = PR[90,1] + 29.952;
   1:  PR[91,2] = PR[90,2] + -31.014;
   1:  PR[91,3] = PR[90,3] + 96.898;
   1:L PR[91] R[100]mm/sec CNT100;
   1:  PR[91,1] = PR[90,1] + 33.821;
   1:  PR[91,2] = PR[90,2] + -30.939;
   1:  PR[91,3] = PR[90,3] + 96.905;
   1:L PR[91] R[100]mm/sec CNT100;
   1:  PR[91,1] = PR[90,1] + 35.643;
   1:  PR[91,2] = PR[90,2] + -30.709;
   1:  PR[91,3] = PR[90,3] + 96.923;
   1:L PR[91] R[100]mm/sec CNT100;
   1:  PR[91,1] = PR[90,1] + 38.961;
   1:  PR[91,2] = PR[90,2] + -30.023;
   1:  PR[91,3] = PR[90,3] + 96.931;
   1:L PR[91] R[100]mm/sec CNT100;
   1:  PR[91,1] = PR[90,1] + 41.137;
   1:  PR[91,2] = PR[90,2] + -29.341;
   1:  PR[91,3] = PR[90,3] + 96.947;
   1:L PR[91] R[100]mm/sec CNT100;
   1:  PR[91,1] = PR[90,1] + 43.729;
   1:  PR[91,2] = PR[90,2] + -28.282;
   1:  PR[91,3] = PR[90,3] + 96.957;
   1:L PR[91] R[100]mm/sec CNT100;
   1:  PR[91,1] = PR[90,1] + 46.218;
   1:  PR[91,2] = PR[90,2] + -26.980;
   1:  PR[91,3] = PR[90,3] + 96.970;
   1:L PR[91] R[100]mm/sec CNT100;
   1:  PR[91,1] = PR[90,1] + 47.983;
   1:  PR[91,2] = PR[90,2] + -25.844;
   1:  PR[91,3] = PR[90,3] + 96.983;
   1:L PR[91] R[100]mm/sec CNT100;
   1:  PR[91,1] = PR[90,1] + 50.702;
   1:  PR[91,2] = PR[90,2] + -23.741;
   1:  PR[91,3] = PR[90,3] + 96.992;
   1:L PR[91] R[100]mm/sec CNT100;
   1:  PR[91,1] = PR[90,1] + 51.627;
   1:  PR[91,2] = PR[90,2] + -22.872;
   1:  PR[91,3] = PR[90,3] + 97.008;
   1:L PR[91] R[100]mm/sec CNT100;
   1:  PR[91,1] = PR[90,1] + 54.429;
   1:  PR[91,2] = PR[90,2] + -19.791;
   1:  PR[91,3] = PR[90,3] + 97.014;
   1:L PR[91] R[100]mm/sec CNT100;
   1:  PR[91,1] = PR[90,1] + 54.623;
   1:  PR[91,2] = PR[90,2] + -19.527;
   1:  PR[91,3] = PR[90,3] + 97.033;
   1:L PR[91] R[100]mm/sec CNT100;
   1:  PR[91,1] = PR[90,1] + 55.950;
   1:  PR[91,2] = PR[90,2] + -17.444;
   1:  PR[91,3] = PR[90,3] + 97.034;
   1:L PR[91] R[100]mm/sec CNT100;
   1:  PR[91,1] = PR[90,1] + 57.287;
   1:  PR[91,2] = PR[90,2] + -15.427;
   1:  PR[91,3] = PR[90,3] + 97.046;
   1:L PR[91] R[100]mm/sec CNT100;
   1:  PR[91,1] = PR[90,1] + 59.343;
   1:  PR[91,2] = PR[90,2] + -10.755;
   1:  PR[91,3] = PR[90,3] + 97.057;
   1:L PR[91] R[100]mm/sec CNT100;
   1:  PR[91,1] = PR[90,1] + 59.644;
   1:  PR[91,2] = PR[90,2] + -9.515;
   1:  PR[91,3] = PR[90,3] + 97.080;
   1:L PR[91] R[100]mm/sec CNT100;
   1:  PR[91,1] = PR[90,1] + 60.584;
   1:  PR[91,2] = PR[90,2] + -5.800;
   1:  PR[91,3] = PR[90,3] + 97.086;
   1:L PR[91] R[100]mm/sec CNT100;
   1:  PR[91,1] = PR[90,1] + 61.001;
   1:  PR[91,2] = PR[90,2] + -0.729;
   1:  PR[91,3] = PR[90,3] + 97.103;
   1:L PR[91] R[100]mm/sec CNT100;
   1:  PR[91,1] = PR[90,1] + 60.584;
   1:  PR[91,2] = PR[90,2] + 4.341;
   1:  PR[91,3] = PR[90,3] + 97.127;
   1:L PR[91] R[100]mm/sec CNT100;
   1:  PR[91,1] = PR[90,1] + 59.644;
   1:  PR[91,2] = PR[90,2] + 8.056;
   1:  PR[91,3] = PR[90,3] + 97.150;
   1:L PR[91] R[100]mm/sec CNT100;
   1:  PR[91,1] = PR[90,1] + 59.343;
   1:  PR[91,2] = PR[90,2] + 9.296;
   1:  PR[91,3] = PR[90,3] + 97.167;
   1:L PR[91] R[100]mm/sec CNT100;
   1:  PR[91,1] = PR[90,1] + 57.287;
   1:  PR[91,2] = PR[90,2] + 13.968;
   1:  PR[91,3] = PR[90,3] + 97.173;
   1:L PR[91] R[100]mm/sec CNT100;
   1:  PR[91,1] = PR[90,1] + 55.950;
   1:  PR[91,2] = PR[90,2] + 15.985;
   1:  PR[91,3] = PR[90,3] + 97.197;
   1:L PR[91] R[100]mm/sec CNT100;
   1:  PR[91,1] = PR[90,1] + 54.623;
   1:  PR[91,2] = PR[90,2] + 18.068;
   1:  PR[91,3] = PR[90,3] + 97.208;
   1:L PR[91] R[100]mm/sec CNT100;
   1:  PR[91,1] = PR[90,1] + 54.429;
   1:  PR[91,2] = PR[90,2] + 18.332;
   1:  PR[91,3] = PR[90,3] + 97.219;
   1:L PR[91] R[100]mm/sec CNT100;
   1:  PR[91,1] = PR[90,1] + 51.627;
   1:  PR[91,2] = PR[90,2] + 21.412;
   1:  PR[91,3] = PR[90,3] + 97.221;
   1:L PR[91] R[100]mm/sec CNT100;
   1:  PR[91,1] = PR[90,1] + 50.703;
   1:  PR[91,2] = PR[90,2] + 22.281;
   1:  PR[91,3] = PR[90,3] + 97.240;
   1:L PR[91] R[100]mm/sec CNT100;
   1:  PR[91,1] = PR[90,1] + 47.984;
   1:  PR[91,2] = PR[90,2] + 24.384;
   1:  PR[91,3] = PR[90,3] + 97.245;
   1:L PR[91] R[100]mm/sec CNT100;
   1:  PR[91,1] = PR[90,1] + 46.221;
   1:  PR[91,2] = PR[90,2] + 25.519;
   1:  PR[91,3] = PR[90,3] + 97.261;
   1:L PR[91] R[100]mm/sec CNT100;
   1:  PR[91,1] = PR[90,1] + 43.733;
   1:  PR[91,2] = PR[90,2] + 26.821;
   1:  PR[91,3] = PR[90,3] + 97.271;
   1:L PR[91] R[100]mm/sec CNT100;
   1:  PR[91,1] = PR[90,1] + 41.141;
   1:  PR[91,2] = PR[90,2] + 27.881;
   1:  PR[91,3] = PR[90,3] + 97.284;
   1:L PR[91] R[100]mm/sec CNT100;
   1:  PR[91,1] = PR[90,1] + 38.967;
   1:  PR[91,2] = PR[90,2] + 28.562;
   1:  PR[91,3] = PR[90,3] + 97.296;
   1:L PR[91] R[100]mm/sec CNT100;
   1:  PR[91,1] = PR[90,1] + 35.650;
   1:  PR[91,2] = PR[90,2] + 29.250;
   1:  PR[91,3] = PR[90,3] + 97.307;
   1:L PR[91] R[100]mm/sec CNT100;
   1:  PR[91,1] = PR[90,1] + 33.828;
   1:  PR[91,2] = PR[90,2] + 29.479;
   1:  PR[91,3] = PR[90,3] + 97.322;
   1:L PR[91] R[100]mm/sec CNT100;
   1:  PR[91,1] = PR[90,1] + 29.961;
   1:  PR[91,2] = PR[90,2] + 29.556;
   1:  PR[91,3] = PR[90,3] + 97.331;
   1:L PR[91] R[100]mm/sec CNT100;
   1:  PR[91,1] = PR[90,1] + 28.489;
   1:  PR[91,2] = PR[90,2] + 29.474;
   1:  PR[91,3] = PR[90,3] + 97.348;
   1:L PR[91] R[100]mm/sec CNT100;
   1:  PR[91,1] = PR[90,1] + 24.336;
   1:  PR[91,2] = PR[90,2] + 28.801;
   1:  PR[91,3] = PR[90,3] + 97.355;
   1:L PR[91] R[100]mm/sec CNT100;
   1:  PR[91,1] = PR[90,1] + 22.553;
   1:  PR[91,2] = PR[90,2] + 28.380;
   1:  PR[91,3] = PR[90,3] + 97.374;
   1:L PR[91] R[100]mm/sec CNT100;
   1:  PR[91,1] = PR[90,1] + 19.478;
   1:  PR[91,2] = PR[90,2] + 28.435;
   1:  PR[91,3] = PR[90,3] + 97.383;
   1:L PR[91] R[100]mm/sec CNT100;
   1:  PR[91,1] = PR[90,1] + 13.914;
   1:  PR[91,2] = PR[90,2] + 28.656;
   1:  PR[91,3] = PR[90,3] + 97.397;
   1:L PR[91] R[100]mm/sec CNT100;
   1:  PR[91,1] = PR[90,1] + 4.658;
   1:  PR[91,2] = PR[90,2] + 28.213;
   1:  PR[91,3] = PR[90,3] + 97.422;
   1:L PR[91] R[100]mm/sec CNT100;
   1:  PR[91,1] = PR[90,1] + -5.612;
   1:  PR[91,2] = PR[90,2] + 27.093;
   1:  PR[91,3] = PR[90,3] + 97.465;
   1:L PR[91] R[100]mm/sec CNT100;
   1:  PR[91,1] = PR[90,1] + -15.183;
   1:  PR[91,2] = PR[90,2] + 25.356;
   1:  PR[91,3] = PR[90,3] + 97.512;
   1:L PR[91] R[100]mm/sec CNT100;
   1:  PR[91,1] = PR[90,1] + -20.066;
   1:  PR[91,2] = PR[90,2] + 24.087;
   1:  PR[91,3] = PR[90,3] + 97.556;
   1:L PR[91] R[100]mm/sec CNT100;
   1:  PR[91,1] = PR[90,1] + -23.878;
   1:  PR[91,2] = PR[90,2] + 23.078;
   1:  PR[91,3] = PR[90,3] + 97.579;
   1:L PR[91] R[100]mm/sec CNT100;
   1:  PR[91,1] = PR[90,1] + -31.581;
   1:  PR[91,2] = PR[90,2] + 20.332;
   1:  PR[91,3] = PR[90,3] + 97.597;
   1:L PR[91] R[100]mm/sec CNT100;
   1:  PR[91,1] = PR[90,1] + -38.178;
   1:  PR[91,2] = PR[90,2] + 17.213;
   1:  PR[91,3] = PR[90,3] + 97.635;
   1:L PR[91] R[100]mm/sec CNT100;
   1:  PR[91,1] = PR[90,1] + -38.338;
   1:  PR[91,2] = PR[90,2] + 17.112;
   1:  PR[91,3] = PR[90,3] + 97.668;
   1:L PR[91] R[100]mm/sec CNT100;
   1:  PR[91,1] = PR[90,1] + -43.000;
   1:  PR[91,2] = PR[90,2] + 13.888;
   1:  PR[91,3] = PR[90,3] + 97.669;
   1:L PR[91] R[100]mm/sec CNT100;
   1:  PR[91] = PR[90];
   1:  PR[91,1] = PR[90,1] + -45.475;
   1:  PR[91,2] = PR[90,2] + 9.692;
   1:  PR[91,3] = PR[90,3] + 98.995;
   1:L PR[91] R[100]mm/sec CNT100;
   1:  PR[91,1] = PR[90,1] + -46.506;
   1:  PR[91,2] = PR[90,2] + 8.278;
   1:  PR[91,3] = PR[90,3] + 97.715;
   1:L PR[91] R[100]mm/sec CNT100;
   1:  PR[91,1] = PR[90,1] + -48.544;
   1:  PR[91,2] = PR[90,2] + 4.636;
   1:  PR[91,3] = PR[90,3] + 97.723;
   1:L PR[91] R[100]mm/sec CNT100;
   1:  PR[91,1] = PR[90,1] + -48.789;
   1:  PR[91,2] = PR[90,2] + 4.059;
   1:  PR[91,3] = PR[90,3] + 97.742;
   1:L PR[91] R[100]mm/sec CNT100;
   1:  PR[91,1] = PR[90,1] + -49.633;
   1:  PR[91,2] = PR[90,2] + -0.522;
   1:  PR[91,3] = PR[90,3] + 97.745;
   1:L PR[91] R[100]mm/sec CNT100;
   1:  PR[91,1] = PR[90,1] + -49.652;
   1:  PR[91,2] = PR[90,2] + -0.655;
   1:  PR[91,3] = PR[90,3] + 97.766;
   1:L PR[91] R[100]mm/sec CNT100;
   1:  PR[91,1] = PR[90,1] + -48.823;
   1:  PR[91,2] = PR[90,2] + -4.526;
   1:  PR[91,3] = PR[90,3] + 97.767;
   1:L PR[91] R[100]mm/sec CNT100;
   1:  PR[91,1] = PR[90,1] + -48.697;
   1:  PR[91,2] = PR[90,2] + -5.464;
   1:  PR[91,3] = PR[90,3] + 97.785;
   1:L PR[91] R[100]mm/sec CNT100;
   1:  PR[91,1] = PR[90,1] + -48.310;
   1:  PR[91,2] = PR[90,2] + -6.384;
   1:  PR[91,3] = PR[90,3] + 97.790;
   1:L PR[91] R[100]mm/sec CNT100;
   1:  PR[91,1] = PR[90,1] + -46.512;
   1:  PR[91,2] = PR[90,2] + -9.602;
   1:  PR[91,3] = PR[90,3] + 97.794;
   1:L PR[91] R[100]mm/sec CNT100;
   1:  PR[91,1] = PR[90,1] + -45.298;
   1:  PR[91,2] = PR[90,2] + -11.285;
   1:  PR[91,3] = PR[90,3] + 97.811;
   1:L PR[91] R[100]mm/sec CNT100;
   1:  PR[91,1] = PR[90,1] + -43.541;
   1:  PR[91,2] = PR[90,2] + -13.068;
   1:  PR[91,3] = PR[90,3] + 97.821;
   1:L PR[91] R[100]mm/sec CNT100;
   1:  PR[91,1] = PR[90,1] + -41.041;
   1:  PR[91,2] = PR[90,2] + -15.464;
   1:  PR[91,3] = PR[90,3] + 97.832;
   1:L PR[91] R[100]mm/sec CNT100;
   1:  PR[91,1] = PR[90,1] + -38.983;
   1:  PR[91,2] = PR[90,2] + -16.899;
   1:  PR[91,3] = PR[90,3] + 97.848;
   1:L PR[91] R[100]mm/sec CNT100;
   1:  PR[91,1] = PR[90,1] + -35.940;
   1:  PR[91,2] = PR[90,2] + -18.820;
   1:  PR[91,3] = PR[90,3] + 97.860;
   1:L PR[91] R[100]mm/sec CNT100;
   1:  PR[91,1] = PR[90,1] + -29.296;
   1:  PR[91,2] = PR[90,2] + -21.964;
   1:  PR[91,3] = PR[90,3] + 97.877;
   1:L PR[91] R[100]mm/sec CNT100;
   1:  PR[91,1] = PR[90,1] + -21.539;
   1:  PR[91,2] = PR[90,2] + -24.732;
   1:  PR[91,3] = PR[90,3] + 97.911;
   1:L PR[91] R[100]mm/sec CNT100;
   1:  PR[91,1] = PR[90,1] + -16.949;
   1:  PR[91,2] = PR[90,2] + -25.948;
   1:  PR[91,3] = PR[90,3] + 97.949;
   1:L PR[91] R[100]mm/sec CNT100;
   1:  PR[91,1] = PR[90,1] + -12.780;
   1:  PR[91,2] = PR[90,2] + -27.031;
   1:  PR[91,3] = PR[90,3] + 97.971;
   1:L PR[91] R[100]mm/sec CNT100;
   1:  PR[91,1] = PR[90,1] + -5.199;
   1:  PR[91,2] = PR[90,2] + -28.417;
   1:  PR[91,3] = PR[90,3] + 97.991;
   1:L PR[91] R[100]mm/sec CNT100;
   1:  PR[91,1] = PR[90,1] + -3.145;
   1:  PR[91,2] = PR[90,2] + -28.783;
   1:  PR[91,3] = PR[90,3] + 98.026;
   1:L PR[91] R[100]mm/sec CNT100;
   1:  PR[91,1] = PR[90,1] + 5.106;
   1:  PR[91,2] = PR[90,2] + -29.684;
   1:  PR[91,3] = PR[90,3] + 98.036;
   1:L PR[91] R[100]mm/sec CNT100;
   1:  PR[91,1] = PR[90,1] + 6.641;
   1:  PR[91,2] = PR[90,2] + -29.893;
   1:  PR[91,3] = PR[90,3] + 98.074;
   1:L PR[91] R[100]mm/sec CNT100;
   1:  PR[91,1] = PR[90,1] + 10.896;
   1:  PR[91,2] = PR[90,2] + -30.120;
   1:  PR[91,3] = PR[90,3] + 98.081;
   1:L PR[91] R[100]mm/sec CNT100;
   1:  PR[91,1] = PR[90,1] + 16.041;
   1:  PR[91,2] = PR[90,2] + -30.372;
   1:  PR[91,3] = PR[90,3] + 98.101;
   1:L PR[91] R[100]mm/sec CNT100;
   1:  PR[91,1] = PR[90,1] + 18.590;
   1:  PR[91,2] = PR[90,2] + -30.271;
   1:  PR[91,3] = PR[90,3] + 98.125;
   1:L PR[91] R[100]mm/sec CNT100;
   1:  PR[91,1] = PR[90,1] + 25.648;
   1:  PR[91,2] = PR[90,2] + -29.896;
   1:  PR[91,3] = PR[90,3] + 98.137;
   1:L PR[91] R[100]mm/sec CNT100;
   1:  PR[91,1] = PR[90,1] + 25.448;
   1:  PR[91,2] = PR[90,2] + -30.607;
   1:  PR[91,3] = PR[90,3] + 98.169;
   1:L PR[91] R[100]mm/sec CNT100;
   1:  PR[91,1] = PR[90,1] + 28.784;
   1:  PR[91,2] = PR[90,2] + -31.148;
   1:  PR[91,3] = PR[90,3] + 98.173;
   1:L PR[91] R[100]mm/sec CNT100;
   1:  PR[91,1] = PR[90,1] + 29.348;
   1:  PR[91,2] = PR[90,2] + -31.179;
   1:  PR[91,3] = PR[90,3] + 98.188;
   1:L PR[91] R[100]mm/sec CNT100;
   1:  PR[91,1] = PR[90,1] + 34.258;
   1:  PR[91,2] = PR[90,2] + -31.084;
   1:  PR[91,3] = PR[90,3] + 98.191;
   1:L PR[91] R[100]mm/sec CNT100;
   1:  PR[91,1] = PR[90,1] + 35.080;
   1:  PR[91,2] = PR[90,2] + -30.981;
   1:  PR[91,3] = PR[90,3] + 98.214;
   1:L PR[91] R[100]mm/sec CNT100;
   1:  PR[91,1] = PR[90,1] + 39.542;
   1:  PR[91,2] = PR[90,2] + -30.057;
   1:  PR[91,3] = PR[90,3] + 98.217;
   1:L PR[91] R[100]mm/sec CNT100;
   1:  PR[91,1] = PR[90,1] + 40.641;
   1:  PR[91,2] = PR[90,2] + -29.713;
   1:  PR[91,3] = PR[90,3] + 98.239;
   1:L PR[91] R[100]mm/sec CNT100;
   1:  PR[91,1] = PR[90,1] + 44.461;
   1:  PR[91,2] = PR[90,2] + -28.152;
   1:  PR[91,3] = PR[90,3] + 98.244;
   1:L PR[91] R[100]mm/sec CNT100;
   1:  PR[91,1] = PR[90,1] + 45.821;
   1:  PR[91,2] = PR[90,2] + -27.441;
   1:  PR[91,3] = PR[90,3] + 98.263;
   1:L PR[91] R[100]mm/sec CNT100;
   1:  PR[91,1] = PR[90,1] + 48.863;
   1:  PR[91,2] = PR[90,2] + -25.483;
   1:  PR[91,3] = PR[90,3] + 98.270;
   1:L PR[91] R[100]mm/sec CNT100;
   1:  PR[91,1] = PR[90,1] + 50.435;
   1:  PR[91,2] = PR[90,2] + -24.267;
   1:  PR[91,3] = PR[90,3] + 98.287;
   1:L PR[91] R[100]mm/sec CNT100;
   1:  PR[91,1] = PR[90,1] + 52.635;
   1:  PR[91,2] = PR[90,2] + -22.198;
   1:  PR[91,3] = PR[90,3] + 98.296;
   1:L PR[91] R[100]mm/sec CNT100;
   1:  PR[91,1] = PR[90,1] + 54.323;
   1:  PR[91,2] = PR[90,2] + -20.343;
   1:  PR[91,3] = PR[90,3] + 98.310;
   1:L PR[91] R[100]mm/sec CNT100;
   1:  PR[91,1] = PR[90,1] + 55.712;
   1:  PR[91,2] = PR[90,2] + -18.450;
   1:  PR[91,3] = PR[90,3] + 98.321;
   1:L PR[91] R[100]mm/sec CNT100;
   1:  PR[91,1] = PR[90,1] + 57.371;
   1:  PR[91,2] = PR[90,2] + -15.845;
   1:  PR[91,3] = PR[90,3] + 98.332;
   1:L PR[91] R[100]mm/sec CNT100;
   1:  PR[91,1] = PR[90,1] + 58.087;
   1:  PR[91,2] = PR[90,2] + -14.370;
   1:  PR[91,3] = PR[90,3] + 98.347;
   1:L PR[91] R[100]mm/sec CNT100;
   1:  PR[91,1] = PR[90,1] + 59.526;
   1:  PR[91,2] = PR[90,2] + -10.971;
   1:  PR[91,3] = PR[90,3] + 98.354;
   1:L PR[91] R[100]mm/sec CNT100;
   1:  PR[91,1] = PR[90,1] + 59.787;
   1:  PR[91,2] = PR[90,2] + -10.029;
   1:  PR[91,3] = PR[90,3] + 98.371;
   1:L PR[91] R[100]mm/sec CNT100;
   1:  PR[91,1] = PR[90,1] + 60.788;
   1:  PR[91,2] = PR[90,2] + -5.902;
   1:  PR[91,3] = PR[90,3] + 98.376;
   1:L PR[91] R[100]mm/sec CNT100;
   1:  PR[91,1] = PR[90,1] + 61.174;
   1:  PR[91,2] = PR[90,2] + -1.109;
   1:  PR[91,3] = PR[90,3] + 98.395;
   1:L PR[91] R[100]mm/sec CNT100;
   1:  PR[91,1] = PR[90,1] + 61.192;
   1:  PR[91,2] = PR[90,2] + -0.755;
   1:  PR[91,3] = PR[90,3] + 98.418;
   1:L PR[91] R[100]mm/sec CNT100;
   1:  PR[91,1] = PR[90,1] + 60.788;
   1:  PR[91,2] = PR[90,2] + 4.445;
   1:  PR[91,3] = PR[90,3] + 98.419;
   1:L PR[91] R[100]mm/sec CNT100;
   1:  PR[91,1] = PR[90,1] + 59.787;
   1:  PR[91,2] = PR[90,2] + 8.570;
   1:  PR[91,3] = PR[90,3] + 98.443;
   1:L PR[91] R[100]mm/sec CNT100;
   1:  PR[91,1] = PR[90,1] + 59.526;
   1:  PR[91,2] = PR[90,2] + 9.512;
   1:  PR[91,3] = PR[90,3] + 98.463;
   1:L PR[91] R[100]mm/sec CNT100;
   1:  PR[91,1] = PR[90,1] + 58.087;
   1:  PR[91,2] = PR[90,2] + 12.910;
   1:  PR[91,3] = PR[90,3] + 98.467;
   1:L PR[91] R[100]mm/sec CNT100;
   1:  PR[91,1] = PR[90,1] + 57.372;
   1:  PR[91,2] = PR[90,2] + 14.385;
   1:  PR[91,3] = PR[90,3] + 98.484;
   1:L PR[91] R[100]mm/sec CNT100;
   1:  PR[91,1] = PR[90,1] + 55.713;
   1:  PR[91,2] = PR[90,2] + 16.990;
   1:  PR[91,3] = PR[90,3] + 98.492;
   1:L PR[91] R[100]mm/sec CNT100;
   1:  PR[91,1] = PR[90,1] + 54.325;
   1:  PR[91,2] = PR[90,2] + 18.882;
   1:  PR[91,3] = PR[90,3] + 98.506;
   1:L PR[91] R[100]mm/sec CNT100;
   1:  PR[91,1] = PR[90,1] + 52.637;
   1:  PR[91,2] = PR[90,2] + 20.737;
   1:  PR[91,3] = PR[90,3] + 98.517;
   1:L PR[91] R[100]mm/sec CNT100;
   1:  PR[91,1] = PR[90,1] + 50.438;
   1:  PR[91,2] = PR[90,2] + 22.806;
   1:  PR[91,3] = PR[90,3] + 98.529;
   1:L PR[91] R[100]mm/sec CNT100;
   1:  PR[91,1] = PR[90,1] + 48.866;
   1:  PR[91,2] = PR[90,2] + 24.022;
   1:  PR[91,3] = PR[90,3] + 98.543;
   1:L PR[91] R[100]mm/sec CNT100;
   1:  PR[91,1] = PR[90,1] + 45.826;
   1:  PR[91,2] = PR[90,2] + 25.979;
   1:  PR[91,3] = PR[90,3] + 98.552;
   1:L PR[91] R[100]mm/sec CNT100;
   1:  PR[91,1] = PR[90,1] + 44.466;
   1:  PR[91,2] = PR[90,2] + 26.691;
   1:  PR[91,3] = PR[90,3] + 98.569;
   1:L PR[91] R[100]mm/sec CNT100;
   1:  PR[91,1] = PR[90,1] + 40.648;
   1:  PR[91,2] = PR[90,2] + 28.252;
   1:  PR[91,3] = PR[90,3] + 98.576;
   1:L PR[91] R[100]mm/sec CNT100;
   1:  PR[91,1] = PR[90,1] + 39.550;
   1:  PR[91,2] = PR[90,2] + 28.596;
   1:  PR[91,3] = PR[90,3] + 98.595;
   1:L PR[91] R[100]mm/sec CNT100;
   1:  PR[91,1] = PR[90,1] + 35.089;
   1:  PR[91,2] = PR[90,2] + 29.521;
   1:  PR[91,3] = PR[90,3] + 98.600;
   1:L PR[91] R[100]mm/sec CNT100;
   1:  PR[91,1] = PR[90,1] + 34.267;
   1:  PR[91,2] = PR[90,2] + 29.624;
   1:  PR[91,3] = PR[90,3] + 98.621;
   1:L PR[91] R[100]mm/sec CNT100;
   1:  PR[91,1] = PR[90,1] + 29.359;
   1:  PR[91,2] = PR[90,2] + 29.721;
   1:  PR[91,3] = PR[90,3] + 98.625;
   1:L PR[91] R[100]mm/sec CNT100;
   1:  PR[91,1] = PR[90,1] + 28.796;
   1:  PR[91,2] = PR[90,2] + 29.690;
   1:  PR[91,3] = PR[90,3] + 98.648;
   1:L PR[91] R[100]mm/sec CNT100;
   1:  PR[91,1] = PR[90,1] + 23.729;
   1:  PR[91,2] = PR[90,2] + 28.869;
   1:  PR[91,3] = PR[90,3] + 98.650;
   1:L PR[91] R[100]mm/sec CNT100;
   1:  PR[91,1] = PR[90,1] + 23.140;
   1:  PR[91,2] = PR[90,2] + 28.730;
   1:  PR[91,3] = PR[90,3] + 98.674;
   1:L PR[91] R[100]mm/sec CNT100;
   1:  PR[91,1] = PR[90,1] + 18.623;
   1:  PR[91,2] = PR[90,2] + 28.811;
   1:  PR[91,3] = PR[90,3] + 98.677;
   1:L PR[91] R[100]mm/sec CNT100;
   1:  PR[91,1] = PR[90,1] + 16.042;
   1:  PR[91,2] = PR[90,2] + 28.913;
   1:  PR[91,3] = PR[90,3] + 98.698;
   1:L PR[91] R[100]mm/sec CNT100;
   1:  PR[91,1] = PR[90,1] + 10.897;
   1:  PR[91,2] = PR[90,2] + 28.661;
   1:  PR[91,3] = PR[90,3] + 98.710;
   1:L PR[91] R[100]mm/sec CNT100;
   1:  PR[91,1] = PR[90,1] + 6.641;
   1:  PR[91,2] = PR[90,2] + 28.434;
   1:  PR[91,3] = PR[90,3] + 98.733;
   1:L PR[91] R[100]mm/sec CNT100;
   1:  PR[91,1] = PR[90,1] + 5.106;
   1:  PR[91,2] = PR[90,2] + 28.225;
   1:  PR[91,3] = PR[90,3] + 98.753;
   1:L PR[91] R[100]mm/sec CNT100;
   1:  PR[91,1] = PR[90,1] + -3.145;
   1:  PR[91,2] = PR[90,2] + 27.325;
   1:  PR[91,3] = PR[90,3] + 98.760;
   1:L PR[91] R[100]mm/sec CNT100;
   1:  PR[91,1] = PR[90,1] + -5.199;
   1:  PR[91,2] = PR[90,2] + 26.959;
   1:  PR[91,3] = PR[90,3] + 98.799;
   1:L PR[91] R[100]mm/sec CNT100;
   1:  PR[91,1] = PR[90,1] + -12.780;
   1:  PR[91,2] = PR[90,2] + 25.572;
   1:  PR[91,3] = PR[90,3] + 98.808;
   1:L PR[91] R[100]mm/sec CNT100;
   1:  PR[91,1] = PR[90,1] + -16.949;
   1:  PR[91,2] = PR[90,2] + 24.489;
   1:  PR[91,3] = PR[90,3] + 98.844;
   1:L PR[91] R[100]mm/sec CNT100;
   1:  PR[91,1] = PR[90,1] + -21.539;
   1:  PR[91,2] = PR[90,2] + 23.273;
   1:  PR[91,3] = PR[90,3] + 98.864;
   1:L PR[91] R[100]mm/sec CNT100;
   1:  PR[91,1] = PR[90,1] + -29.296;
   1:  PR[91,2] = PR[90,2] + 20.506;
   1:  PR[91,3] = PR[90,3] + 98.886;
   1:L PR[91] R[100]mm/sec CNT100;
   1:  PR[91,1] = PR[90,1] + -35.940;
   1:  PR[91,2] = PR[90,2] + 17.361;
   1:  PR[91,3] = PR[90,3] + 98.924;
   1:L PR[91] R[100]mm/sec CNT100;
   1:  PR[91,1] = PR[90,1] + -38.987;
   1:  PR[91,2] = PR[90,2] + 15.439;
   1:  PR[91,3] = PR[90,3] + 98.958;
   1:L PR[91] R[100]mm/sec CNT100;
   1:  PR[91,1] = PR[90,1] + -41.065;
   1:  PR[91,2] = PR[90,2] + 14.002;
   1:  PR[91,3] = PR[90,3] + 98.974;
   1:L PR[91] R[100]mm/sec CNT100;
   1:  PR[91,1] = PR[90,1] + -42.431;
   1:  PR[91,2] = PR[90,2] + 12.638;
   1:  PR[91,3] = PR[90,3] + 98.986;
   1:L PR[91] R[100]mm/sec CNT100;
   1:  PR[91] = PR[90];
   1:  PR[91,1] = PR[90,1] + -44.925;
   1:  PR[91,2] = PR[90,2] + 7.871;
   1:  PR[91,3] = PR[90,3] + 100.295;
   1:L PR[91] R[100]mm/sec CNT100;
   1:  PR[91,1] = PR[90,1] + -46.371;
   1:  PR[91,2] = PR[90,2] + 5.287;
   1:  PR[91,3] = PR[90,3] + 99.008;
   1:L PR[91] R[100]mm/sec CNT100;
   1:  PR[91,1] = PR[90,1] + -46.992;
   1:  PR[91,2] = PR[90,2] + 3.826;
   1:  PR[91,3] = PR[90,3] + 99.021;
   1:L PR[91] R[100]mm/sec CNT100;
   1:  PR[91,1] = PR[90,1] + -47.631;
   1:  PR[91,2] = PR[90,2] + 0.359;
   1:  PR[91,3] = PR[90,3] + 99.029;
   1:L PR[91] R[100]mm/sec CNT100;
   1:  PR[91,1] = PR[90,1] + -47.771;
   1:  PR[91,2] = PR[90,2] + -0.655;
   1:  PR[91,3] = PR[90,3] + 99.045;
   1:L PR[91] R[100]mm/sec CNT100;
   1:  PR[91,1] = PR[90,1] + -47.136;
   1:  PR[91,2] = PR[90,2] + -3.623;
   1:  PR[91,3] = PR[90,3] + 99.050;
   1:L PR[91] R[100]mm/sec CNT100;
   1:  PR[91,1] = PR[90,1] + -46.916;
   1:  PR[91,2] = PR[90,2] + -5.255;
   1:  PR[91,3] = PR[90,3] + 99.064;
   1:L PR[91] R[100]mm/sec CNT100;
   1:  PR[91,1] = PR[90,1] + -46.201;
   1:  PR[91,2] = PR[90,2] + -6.956;
   1:  PR[91,3] = PR[90,3] + 99.072;
   1:L PR[91] R[100]mm/sec CNT100;
   1:  PR[91,1] = PR[90,1] + -44.928;
   1:  PR[91,2] = PR[90,2] + -9.234;
   1:  PR[91,3] = PR[90,3] + 99.081;
   1:L PR[91] R[100]mm/sec CNT100;
   1:  PR[91,1] = PR[90,1] + -43.216;
   1:  PR[91,2] = PR[90,2] + -11.609;
   1:  PR[91,3] = PR[90,3] + 99.093;
   1:L PR[91] R[100]mm/sec CNT100;
   1:  PR[91,1] = PR[90,1] + -42.222;
   1:  PR[91,2] = PR[90,2] + -12.617;
   1:  PR[91,3] = PR[90,3] + 99.106;
   1:L PR[91] R[100]mm/sec CNT100;
   1:  PR[91,1] = PR[90,1] + -39.392;
   1:  PR[91,2] = PR[90,2] + -15.330;
   1:  PR[91,3] = PR[90,3] + 99.113;
   1:L PR[91] R[100]mm/sec CNT100;
   1:  PR[91,1] = PR[90,1] + -39.188;
   1:  PR[91,2] = PR[90,2] + -15.505;
   1:  PR[91,3] = PR[90,3] + 99.131;
   1:L PR[91] R[100]mm/sec CNT100;
   1:  PR[91,1] = PR[90,1] + -33.702;
   1:  PR[91,2] = PR[90,2] + -18.967;
   1:  PR[91,3] = PR[90,3] + 99.133;
   1:L PR[91] R[100]mm/sec CNT100;
   1:  PR[91,1] = PR[90,1] + -27.011;
   1:  PR[91,2] = PR[90,2] + -22.137;
   1:  PR[91,3] = PR[90,3] + 99.163;
   1:L PR[91] R[100]mm/sec CNT100;
   1:  PR[91,1] = PR[90,1] + -19.200;
   1:  PR[91,2] = PR[90,2] + -24.928;
   1:  PR[91,3] = PR[90,3] + 99.197;
   1:L PR[91] R[100]mm/sec CNT100;
   1:  PR[91,1] = PR[90,1] + -13.832;
   1:  PR[91,2] = PR[90,2] + -26.349;
   1:  PR[91,3] = PR[90,3] + 99.236;
   1:L PR[91] R[100]mm/sec CNT100;
   1:  PR[91,1] = PR[90,1] + -10.380;
   1:  PR[91,2] = PR[90,2] + -27.246;
   1:  PR[91,3] = PR[90,3] + 99.262;
   1:L PR[91] R[100]mm/sec CNT100;
   1:  PR[91,1] = PR[90,1] + -0.670;
   1:  PR[91,2] = PR[90,2] + -29.016;
   1:  PR[91,3] = PR[90,3] + 99.279;
   1:L PR[91] R[100]mm/sec CNT100;
   1:  PR[91,1] = PR[90,1] + 4.458;
   1:  PR[91,2] = PR[90,2] + -29.576;
   1:  PR[91,3] = PR[90,3] + 99.325;
   1:L PR[91] R[100]mm/sec CNT100;
   1:  PR[91,1] = PR[90,1] + 8.317;
   1:  PR[91,2] = PR[90,2] + -30.101;
   1:  PR[91,3] = PR[90,3] + 99.349;
   1:L PR[91] R[100]mm/sec CNT100;
   1:  PR[91,1] = PR[90,1] + 18.123;
   1:  PR[91,2] = PR[90,2] + -30.626;
   1:  PR[91,3] = PR[90,3] + 99.367;
   1:L PR[91] R[100]mm/sec CNT100;
   1:  PR[91,1] = PR[90,1] + 26.250;
   1:  PR[91,2] = PR[90,2] + -30.195;
   1:  PR[91,3] = PR[90,3] + 99.413;
   1:L PR[91] R[100]mm/sec CNT100;
   1:  PR[91,1] = PR[90,1] + 26.060;
   1:  PR[91,2] = PR[90,2] + -30.872;
   1:  PR[91,3] = PR[90,3] + 99.451;
   1:L PR[91] R[100]mm/sec CNT100;
   1:  PR[91,1] = PR[90,1] + 28.993;
   1:  PR[91,2] = PR[90,2] + -31.346;
   1:  PR[91,3] = PR[90,3] + 99.454;
   1:L PR[91] R[100]mm/sec CNT100;
   1:  PR[91,1] = PR[90,1] + 34.620;
   1:  PR[91,2] = PR[90,2] + -31.231;
   1:  PR[91,3] = PR[90,3] + 99.468;
   1:L PR[91] R[100]mm/sec CNT100;
   1:  PR[91,1] = PR[90,1] + 40.124;
   1:  PR[91,2] = PR[90,2] + -30.092;
   1:  PR[91,3] = PR[90,3] + 99.494;
   1:L PR[91] R[100]mm/sec CNT100;
   1:  PR[91,1] = PR[90,1] + 40.146;
   1:  PR[91,2] = PR[90,2] + -30.085;
   1:  PR[91,3] = PR[90,3] + 99.521;
   1:L PR[91] R[100]mm/sec CNT100;
   1:  PR[91,1] = PR[90,1] + 45.193;
   1:  PR[91,2] = PR[90,2] + -28.023;
   1:L PR[91] R[100]mm/sec CNT100;
   1:  PR[91,1] = PR[90,1] + 45.424;
   1:  PR[91,2] = PR[90,2] + -27.902;
   1:  PR[91,3] = PR[90,3] + 99.546;
   1:L PR[91] R[100]mm/sec CNT100;
   1:  PR[91,1] = PR[90,1] + 49.743;
   1:  PR[91,2] = PR[90,2] + -25.122;
   1:  PR[91,3] = PR[90,3] + 99.547;
   1:L PR[91] R[100]mm/sec CNT100;
   1:  PR[91,1] = PR[90,1] + 50.169;
   1:  PR[91,2] = PR[90,2] + -24.793;
   1:  PR[91,3] = PR[90,3] + 99.571;
   1:L PR[91] R[100]mm/sec CNT100;
   1:  PR[91,1] = PR[90,1] + 53.644;
   1:  PR[91,2] = PR[90,2] + -21.525;
   1:  PR[91,3] = PR[90,3] + 99.574;
   1:L PR[91] R[100]mm/sec CNT100;
   1:  PR[91,1] = PR[90,1] + 54.218;
   1:  PR[91,2] = PR[90,2] + -20.895;
   1:  PR[91,3] = PR[90,3] + 99.596;
   1:L PR[91] R[100]mm/sec CNT100;
   1:  PR[91,1] = PR[90,1] + 56.802;
   1:  PR[91,2] = PR[90,2] + -17.374;
   1:  PR[91,3] = PR[90,3] + 99.600;
   1:L PR[91] R[100]mm/sec CNT100;
   1:  PR[91,1] = PR[90,1] + 57.445;
   1:  PR[91,2] = PR[90,2] + -16.364;
   1:  PR[91,3] = PR[90,3] + 99.620;
   1:L PR[91] R[100]mm/sec CNT100;
   1:  PR[91,1] = PR[90,1] + 59.170;
   1:  PR[91,2] = PR[90,2] + -12.806;
   1:  PR[91,3] = PR[90,3] + 99.626;
   1:L PR[91] R[100]mm/sec CNT100;
   1:  PR[91,1] = PR[90,1] + 59.773;
   1:  PR[91,2] = PR[90,2] + -11.383;
   1:  PR[91,3] = PR[90,3] + 99.645;
   1:L PR[91] R[100]mm/sec CNT100;
   1:  PR[91,1] = PR[90,1] + 60.727;
   1:  PR[91,2] = PR[90,2] + -7.931;
   1:  PR[91,3] = PR[90,3] + 99.652;
   1:L PR[91] R[100]mm/sec CNT100;
   1:  PR[91,1] = PR[90,1] + 61.163;
   1:  PR[91,2] = PR[90,2] + -6.135;
   1:  PR[91,3] = PR[90,3] + 99.668;
   1:L PR[91] R[100]mm/sec CNT100;
   1:  PR[91,1] = PR[90,1] + 61.350;
   1:  PR[91,2] = PR[90,2] + -3.722;
   1:  PR[91,3] = PR[90,3] + 99.677;
   1:L PR[91] R[100]mm/sec CNT100;
   1:  PR[91,1] = PR[90,1] + 61.612;
   1:  PR[91,2] = PR[90,2] + -0.718;
   1:  PR[91,3] = PR[90,3] + 99.688;
   1:L PR[91] R[100]mm/sec CNT100;
   1:  PR[91,1] = PR[90,1] + 61.475;
   1:  PR[91,2] = PR[90,2] + 1.093;
   1:  PR[91,3] = PR[90,3] + 99.702;
   1:L PR[91] R[100]mm/sec CNT100;
   1:  PR[91,1] = PR[90,1] + 61.166;
   1:  PR[91,2] = PR[90,2] + 4.666;
   1:  PR[91,3] = PR[90,3] + 99.711;
   1:L PR[91] R[100]mm/sec CNT100;
   1:  PR[91,1] = PR[90,1] + 60.727;
   1:  PR[91,2] = PR[90,2] + 6.472;
   1:  PR[91,3] = PR[90,3] + 99.728;
   1:L PR[91] R[100]mm/sec CNT100;
   1:  PR[91,1] = PR[90,1] + 59.774;
   1:  PR[91,2] = PR[90,2] + 9.922;
   1:  PR[91,3] = PR[90,3] + 99.736;
   1:L PR[91] R[100]mm/sec CNT100;
   1:  PR[91,1] = PR[90,1] + 59.171;
   1:  PR[91,2] = PR[90,2] + 11.346;
   1:  PR[91,3] = PR[90,3] + 99.753;
   1:L PR[91] R[100]mm/sec CNT100;
   1:  PR[91,1] = PR[90,1] + 57.446;
   1:  PR[91,2] = PR[90,2] + 14.902;
   1:  PR[91,3] = PR[90,3] + 99.760;
   1:L PR[91] R[100]mm/sec CNT100;
   1:  PR[91,1] = PR[90,1] + 56.803;
   1:  PR[91,2] = PR[90,2] + 15.912;
   1:  PR[91,3] = PR[90,3] + 99.779;
   1:L PR[91] R[100]mm/sec CNT100;
   1:  PR[91,1] = PR[90,1] + 54.221;
   1:  PR[91,2] = PR[90,2] + 19.433;
   1:  PR[91,3] = PR[90,3] + 99.784;
   1:L PR[91] R[100]mm/sec CNT100;
   1:  PR[91,1] = PR[90,1] + 53.647;
   1:  PR[91,2] = PR[90,2] + 20.063;
   1:  PR[91,3] = PR[90,3] + 99.805;
   1:L PR[91] R[100]mm/sec CNT100;
   1:  PR[91,1] = PR[90,1] + 50.174;
   1:  PR[91,2] = PR[90,2] + 23.330;
   1:  PR[91,3] = PR[90,3] + 99.809;
   1:L PR[91] R[100]mm/sec CNT100;
   1:  PR[91,1] = PR[90,1] + 49.748;
   1:  PR[91,2] = PR[90,2] + 23.660;
   1:  PR[91,3] = PR[90,3] + 99.831;
   1:L PR[91] R[100]mm/sec CNT100;
   1:  PR[91,1] = PR[90,1] + 45.431;
   1:  PR[91,2] = PR[90,2] + 26.439;
   1:  PR[91,3] = PR[90,3] + 99.833;
   1:L PR[91] R[100]mm/sec CNT100;
   1:  PR[91,1] = PR[90,1] + 45.200;
   1:  PR[91,2] = PR[90,2] + 26.560;
   1:  PR[91,3] = PR[90,3] + 99.857;
   1:L PR[91] R[100]mm/sec CNT100;
   1:  PR[91,1] = PR[90,1] + 40.155;
   1:  PR[91,2] = PR[90,2] + 28.623;
   1:  PR[91,3] = PR[90,3] + 99.859;
   1:L PR[91] R[100]mm/sec CNT100;
   1:  PR[91,1] = PR[90,1] + 40.133;
   1:  PR[91,2] = PR[90,2] + 28.630;
   1:  PR[91,3] = PR[90,3] + 99.884;
   1:L PR[91] R[100]mm/sec CNT100;
   1:  PR[91,1] = PR[90,1] + 34.626;
   1:  PR[91,2] = PR[90,2] + 29.771;
   1:L PR[91] R[100]mm/sec CNT100;
   1:  PR[91,1] = PR[90,1] + 29.012;
   1:  PR[91,2] = PR[90,2] + 29.888;
   1:  PR[91,3] = PR[90,3] + 99.910;
   1:L PR[91] R[100]mm/sec CNT100;
   1:  PR[91,1] = PR[90,1] + 28.964;
   1:  PR[91,2] = PR[90,2] + 29.884;
   1:  PR[91,3] = PR[90,3] + 99.937;
   1:L PR[91] R[100]mm/sec CNT100;
   1:  PR[91,1] = PR[90,1] + 23.663;
   1:  PR[91,2] = PR[90,2] + 29.025;
   1:L PR[91] R[100]mm/sec CNT100;
   1:  PR[91,1] = PR[90,1] + 18.121;
   1:  PR[91,2] = PR[90,2] + 29.168;
   1:  PR[91,3] = PR[90,3] + 99.962;
   1:L PR[91] R[100]mm/sec CNT100;
   1:  PR[91,1] = PR[90,1] + 8.318;
   1:  PR[91,2] = PR[90,2] + 28.642;
   1:  PR[91,3] = PR[90,3] + 99.988;
   1:L PR[91] R[100]mm/sec CNT100;
   1:  PR[91,1] = PR[90,1] + 4.458;
   1:  PR[91,2] = PR[90,2] + 28.117;
   1:  PR[91,3] = PR[90,3] + 100.034;
   1:L PR[91] R[100]mm/sec CNT100;
   1:  PR[91,1] = PR[90,1] + -0.670;
   1:  PR[91,2] = PR[90,2] + 27.557;
   1:  PR[91,3] = PR[90,3] + 100.052;
   1:L PR[91] R[100]mm/sec CNT100;
   1:  PR[91,1] = PR[90,1] + -10.380;
   1:  PR[91,2] = PR[90,2] + 25.788;
   1:  PR[91,3] = PR[90,3] + 100.076;
   1:L PR[91] R[100]mm/sec CNT100;
   1:  PR[91,1] = PR[90,1] + -13.831;
   1:  PR[91,2] = PR[90,2] + 24.891;
   1:  PR[91,3] = PR[90,3] + 100.122;
   1:L PR[91] R[100]mm/sec CNT100;
   1:  PR[91,1] = PR[90,1] + -19.200;
   1:  PR[91,2] = PR[90,2] + 23.469;
   1:  PR[91,3] = PR[90,3] + 100.139;
   1:L PR[91] R[100]mm/sec CNT100;
   1:  PR[91,1] = PR[90,1] + -27.011;
   1:  PR[91,2] = PR[90,2] + 20.679;
   1:  PR[91,3] = PR[90,3] + 100.165;
   1:L PR[91] R[100]mm/sec CNT100;
   1:  PR[91,1] = PR[90,1] + -33.702;
   1:  PR[91,2] = PR[90,2] + 17.508;
   1:  PR[91,3] = PR[90,3] + 100.203;
   1:L PR[91] R[100]mm/sec CNT100;
   1:  PR[91,1] = PR[90,1] + -39.188;
   1:  PR[91,2] = PR[90,2] + 14.047;
   1:  PR[91,3] = PR[90,3] + 100.238;
   1:L PR[91] R[100]mm/sec CNT100;
   1:  PR[91,1] = PR[90,1] + -39.388;
   1:  PR[91,2] = PR[90,2] + 13.874;
   1:  PR[91,3] = PR[90,3] + 100.268;
   1:L PR[91] R[100]mm/sec CNT100;
   1:  PR[91,1] = PR[90,1] + -43.328;
   1:  PR[91,2] = PR[90,2] + 10.061;
   1:  PR[91,3] = PR[90,3] + 100.269;
   1:L PR[91] R[100]mm/sec CNT100;
   1:  PR[91] = PR[90];
   1:  PR[91,1] = PR[90,1] + -43.344;
   1:  PR[91,2] = PR[90,2] + 7.465;
   1:  PR[91,3] = PR[90,3] + 101.595;
   1:L PR[91] R[100]mm/sec CNT100;
   1:  PR[91,1] = PR[90,1] + -44.199;
   1:  PR[91,2] = PR[90,2] + 5.937;
   1:  PR[91,3] = PR[90,3] + 100.312;
   1:L PR[91] R[100]mm/sec CNT100;
   1:  PR[91,1] = PR[90,1] + -45.194;
   1:  PR[91,2] = PR[90,2] + 3.593;
   1:  PR[91,3] = PR[90,3] + 100.321;
   1:L PR[91] R[100]mm/sec CNT100;
   1:  PR[91,1] = PR[90,1] + -45.628;
   1:  PR[91,2] = PR[90,2] + 1.240;
   1:  PR[91,3] = PR[90,3] + 100.333;
   1:L PR[91] R[100]mm/sec CNT100;
   1:  PR[91,1] = PR[90,1] + -45.891;
   1:  PR[91,2] = PR[90,2] + -0.655;
   1:  PR[91,3] = PR[90,3] + 100.344;
   1:L PR[91] R[100]mm/sec CNT100;
   1:  PR[91,1] = PR[90,1] + -45.449;
   1:  PR[91,2] = PR[90,2] + -2.720;
   1:  PR[91,3] = PR[90,3] + 100.353;
   1:L PR[91] R[100]mm/sec CNT100;
   1:  PR[91,1] = PR[90,1] + -45.135;
   1:  PR[91,2] = PR[90,2] + -5.045;
   1:  PR[91,3] = PR[90,3] + 100.363;
   1:L PR[91] R[100]mm/sec CNT100;
   1:  PR[91,1] = PR[90,1] + -44.092;
   1:  PR[91,2] = PR[90,2] + -7.528;
   1:  PR[91,3] = PR[90,3] + 100.374;
   1:L PR[91] R[100]mm/sec CNT100;
   1:  PR[91,1] = PR[90,1] + -43.344;
   1:  PR[91,2] = PR[90,2] + -8.866;
   1:  PR[91,3] = PR[90,3] + 100.387;
   1:L PR[91] R[100]mm/sec CNT100;
   1:  PR[91,1] = PR[90,1] + -41.134;
   1:  PR[91,2] = PR[90,2] + -11.932;
   1:  PR[91,3] = PR[90,3] + 100.394;
   1:L PR[91] R[100]mm/sec CNT100;
   1:  PR[91,1] = PR[90,1] + -40.904;
   1:  PR[91,2] = PR[90,2] + -12.166;
   1:  PR[91,3] = PR[90,3] + 100.412;
   1:L PR[91] R[100]mm/sec CNT100;
   1:  PR[91,1] = PR[90,1] + -40.040;
   1:  PR[91,2] = PR[90,2] + -12.993;
   1:  PR[91,3] = PR[90,3] + 100.413;
   1:L PR[91] R[100]mm/sec CNT100;
   1:  PR[91,1] = PR[90,1] + -36.989;
   1:  PR[91,2] = PR[90,2] + -15.626;
   1:  PR[91,3] = PR[90,3] + 100.419;
   1:L PR[91] R[100]mm/sec CNT100;
   1:  PR[91,1] = PR[90,1] + -31.464;
   1:  PR[91,2] = PR[90,2] + -19.115;
   1:  PR[91,3] = PR[90,3] + 100.438;
   1:L PR[91] R[100]mm/sec CNT100;
   1:  PR[91,1] = PR[90,1] + -24.726;
   1:  PR[91,2] = PR[90,2] + -22.310;
   1:  PR[91,3] = PR[90,3] + 100.469;
   1:L PR[91] R[100]mm/sec CNT100;
   1:  PR[91,1] = PR[90,1] + -16.862;
   1:  PR[91,2] = PR[90,2] + -25.123;
   1:  PR[91,3] = PR[90,3] + 100.504;
   1:L PR[91] R[100]mm/sec CNT100;
   1:  PR[91,1] = PR[90,1] + -7.975;
   1:  PR[91,2] = PR[90,2] + -27.463;
   1:  PR[91,3] = PR[90,3] + 100.543;
   1:L PR[91] R[100]mm/sec CNT100;
   1:  PR[91,1] = PR[90,1] + 1.801;
   1:  PR[91,2] = PR[90,2] + -29.248;
   1:  PR[91,3] = PR[90,3] + 100.586;
   1:L PR[91] R[100]mm/sec CNT100;
   1:  PR[91,1] = PR[90,1] + 3.810;
   1:  PR[91,2] = PR[90,2] + -29.467;
   1:  PR[91,3] = PR[90,3] + 100.633;
   1:L PR[91] R[100]mm/sec CNT100;
   1:  PR[91,1] = PR[90,1] + 9.993;
   1:  PR[91,2] = PR[90,2] + -30.309;
   1:  PR[91,3] = PR[90,3] + 100.643;
   1:L PR[91] R[100]mm/sec CNT100;
   1:  PR[91,1] = PR[90,1] + 17.071;
   1:  PR[91,2] = PR[90,2] + -30.686;
   1:  PR[91,3] = PR[90,3] + 100.672;
   1:L PR[91] R[100]mm/sec CNT100;
   1:  PR[91,1] = PR[90,1] + 19.711;
   1:  PR[91,2] = PR[90,2] + -30.859;
   1:  PR[91,3] = PR[90,3] + 100.706;
   1:L PR[91] R[100]mm/sec CNT100;
   1:  PR[91,1] = PR[90,1] + 19.899;
   1:  PR[91,2] = PR[90,2] + -30.862;
   1:  PR[91,3] = PR[90,3] + 100.718;
   1:L PR[91] R[100]mm/sec CNT100;
   1:  PR[91,1] = PR[90,1] + 26.852;
   1:  PR[91,2] = PR[90,2] + -30.493;
   1:  PR[91,3] = PR[90,3] + 100.719;
   1:L PR[91] R[100]mm/sec CNT100;
   1:  PR[91,1] = PR[90,1] + 26.671;
   1:  PR[91,2] = PR[90,2] + -31.138;
   1:  PR[91,3] = PR[90,3] + 100.752;
   1:L PR[91] R[100]mm/sec CNT100;
   1:  PR[91,1] = PR[90,1] + 28.452;
   1:  PR[91,2] = PR[90,2] + -31.427;
   1:  PR[91,3] = PR[90,3] + 100.755;
   1:L PR[91] R[100]mm/sec CNT100;
   1:  PR[91,1] = PR[90,1] + 28.695;
   1:  PR[91,2] = PR[90,2] + -31.455;
   1:  PR[91,3] = PR[90,3] + 100.764;
   1:L PR[91] R[100]mm/sec CNT100;
   1:  PR[91,1] = PR[90,1] + 29.671;
   1:  PR[91,2] = PR[90,2] + -31.519;
   1:  PR[91,3] = PR[90,3] + 100.765;
   1:L PR[91] R[100]mm/sec CNT100;
   1:  PR[91,1] = PR[90,1] + 34.356;
   1:  PR[91,2] = PR[90,2] + -31.423;
   1:  PR[91,3] = PR[90,3] + 100.769;
   1:L PR[91] R[100]mm/sec CNT100;
   1:  PR[91,1] = PR[90,1] + 35.246;
   1:  PR[91,2] = PR[90,2] + -31.332;
   1:  PR[91,3] = PR[90,3] + 100.791;
   1:L PR[91] R[100]mm/sec CNT100;
   1:  PR[91,1] = PR[90,1] + 39.887;
   1:  PR[91,2] = PR[90,2] + -30.361;
   1:  PR[91,3] = PR[90,3] + 100.796;
   1:L PR[91] R[100]mm/sec CNT100;
   1:  PR[91,1] = PR[90,1] + 40.682;
   1:  PR[91,2] = PR[90,2] + -30.139;
   1:  PR[91,3] = PR[90,3] + 100.818;
   1:L PR[91] R[100]mm/sec CNT100;
   1:  PR[91,1] = PR[90,1] + 45.128;
   1:  PR[91,2] = PR[90,2] + -28.305;
   1:  PR[91,3] = PR[90,3] + 100.822;
   1:L PR[91] R[100]mm/sec CNT100;
   1:  PR[91,1] = PR[90,1] + 45.801;
   1:  PR[91,2] = PR[90,2] + -27.987;
   1:  PR[91,3] = PR[90,3] + 100.845;
   1:L PR[91] R[100]mm/sec CNT100;
   1:  PR[91,1] = PR[90,1] + 49.908;
   1:  PR[91,2] = PR[90,2] + -25.320;
   1:  PR[91,3] = PR[90,3] + 100.848;
   1:L PR[91] R[100]mm/sec CNT100;
   1:  PR[91,1] = PR[90,1] + 50.441;
   1:  PR[91,2] = PR[90,2] + -24.946;
   1:  PR[91,3] = PR[90,3] + 100.871;
   1:L PR[91] R[100]mm/sec CNT100;
   1:  PR[91,1] = PR[90,1] + 54.067;
   1:  PR[91,2] = PR[90,2] + -21.507;
   1:  PR[91,3] = PR[90,3] + 100.874;
   1:L PR[91] R[100]mm/sec CNT100;
   1:  PR[91,1] = PR[90,1] + 54.453;
   1:  PR[91,2] = PR[90,2] + -21.125;
   1:  PR[91,3] = PR[90,3] + 100.898;
   1:L PR[91] R[100]mm/sec CNT100;
   1:  PR[91,1] = PR[90,1] + 57.716;
   1:  PR[91,2] = PR[90,2] + -16.629;
   1:  PR[91,3] = PR[90,3] + 100.900;
   1:L PR[91] R[100]mm/sec CNT100;
   1:  PR[91,1] = PR[90,1] + 60.117;
   1:  PR[91,2] = PR[90,2] + -11.632;
   1:  PR[91,3] = PR[90,3] + 100.927;
   1:L PR[91] R[100]mm/sec CNT100;
   1:  PR[91,1] = PR[90,1] + 61.589;
   1:  PR[91,2] = PR[90,2] + -6.270;
   1:  PR[91,3] = PR[90,3] + 100.953;
   1:L PR[91] R[100]mm/sec CNT100;
   1:  PR[91,1] = PR[90,1] + 62.101;
   1:  PR[91,2] = PR[90,2] + -0.729;
   1:  PR[91,3] = PR[90,3] + 100.979;
   1:L PR[91] R[100]mm/sec CNT100;
   1:  PR[91,1] = PR[90,1] + 61.589;
   1:  PR[91,2] = PR[90,2] + 4.810;
   1:  PR[91,3] = PR[90,3] + 101.005;
   1:L PR[91] R[100]mm/sec CNT100;
   1:  PR[91,1] = PR[90,1] + 60.117;
   1:  PR[91,2] = PR[90,2] + 10.174;
   1:  PR[91,3] = PR[90,3] + 101.031;
   1:L PR[91] R[100]mm/sec CNT100;
   1:  PR[91,1] = PR[90,1] + 59.976;
   1:  PR[91,2] = PR[90,2] + 10.471;
   1:  PR[91,3] = PR[90,3] + 101.058;
   1:L PR[91] R[100]mm/sec CNT100;
   1:  PR[91,1] = PR[90,1] + 57.718;
   1:  PR[91,2] = PR[90,2] + 15.167;
   1:  PR[91,3] = PR[90,3] + 101.059;
   1:L PR[91] R[100]mm/sec CNT100;
   1:  PR[91,1] = PR[90,1] + 54.455;
   1:  PR[91,2] = PR[90,2] + 19.663;
   1:  PR[91,3] = PR[90,3] + 101.084;
   1:L PR[91] R[100]mm/sec CNT100;
   1:  PR[91,1] = PR[90,1] + 54.070;
   1:  PR[91,2] = PR[90,2] + 20.045;
   1:  PR[91,3] = PR[90,3] + 101.110;
   1:L PR[91] R[100]mm/sec CNT100;
   1:  PR[91,1] = PR[90,1] + 50.445;
   1:  PR[91,2] = PR[90,2] + 23.485;
   1:  PR[91,3] = PR[90,3] + 101.112;
   1:L PR[91] R[100]mm/sec CNT100;
   1:  PR[91,1] = PR[90,1] + 49.912;
   1:  PR[91,2] = PR[90,2] + 23.858;
   1:  PR[91,3] = PR[90,3] + 101.136;
   1:L PR[91] R[100]mm/sec CNT100;
   1:  PR[91,1] = PR[90,1] + 45.805;
   1:  PR[91,2] = PR[90,2] + 26.526;
   1:  PR[91,3] = PR[90,3] + 101.139;
   1:L PR[91] R[100]mm/sec CNT100;
   1:  PR[91,1] = PR[90,1] + 45.133;
   1:  PR[91,2] = PR[90,2] + 26.844;
   1:  PR[91,3] = PR[90,3] + 101.162;
   1:L PR[91] R[100]mm/sec CNT100;
   1:  PR[91,1] = PR[90,1] + 40.687;
   1:  PR[91,2] = PR[90,2] + 28.679;
   1:  PR[91,3] = PR[90,3] + 101.166;
   1:L PR[91] R[100]mm/sec CNT100;
   1:  PR[91,1] = PR[90,1] + 39.892;
   1:  PR[91,2] = PR[90,2] + 28.900;
   1:  PR[91,3] = PR[90,3] + 101.188;
   1:L PR[91] R[100]mm/sec CNT100;
   1:  PR[91,1] = PR[90,1] + 35.251;
   1:  PR[91,2] = PR[90,2] + 29.873;
   1:  PR[91,3] = PR[90,3] + 101.192;
   1:L PR[91] R[100]mm/sec CNT100;
   1:  PR[91,1] = PR[90,1] + 34.362;
   1:  PR[91,2] = PR[90,2] + 29.964;
   1:  PR[91,3] = PR[90,3] + 101.215;
   1:L PR[91] R[100]mm/sec CNT100;
   1:  PR[91,1] = PR[90,1] + 29.677;
   1:  PR[91,2] = PR[90,2] + 30.061;
   1:  PR[91,3] = PR[90,3] + 101.219;
   1:L PR[91] R[100]mm/sec CNT100;
   1:  PR[91,1] = PR[90,1] + 28.703;
   1:  PR[91,2] = PR[90,2] + 29.996;
   1:  PR[91,3] = PR[90,3] + 101.241;
   1:L PR[91] R[100]mm/sec CNT100;
   1:  PR[91,1] = PR[90,1] + 28.411;
   1:  PR[91,2] = PR[90,2] + 29.962;
   1:  PR[91,3] = PR[90,3] + 101.245;
   1:L PR[91] R[100]mm/sec CNT100;
   1:  PR[91,1] = PR[90,1] + 24.273;
   1:  PR[91,2] = PR[90,2] + 29.292;
   1:  PR[91,3] = PR[90,3] + 101.247;
   1:L PR[91] R[100]mm/sec CNT100;
   1:  PR[91,1] = PR[90,1] + 19.975;
   1:  PR[91,2] = PR[90,2] + 29.404;
   1:  PR[91,3] = PR[90,3] + 101.267;
   1:L PR[91] R[100]mm/sec CNT100;
   1:  PR[91,1] = PR[90,1] + 19.713;
   1:  PR[91,2] = PR[90,2] + 29.400;
   1:  PR[91,3] = PR[90,3] + 101.287;
   1:L PR[91] R[100]mm/sec CNT100;
   1:  PR[91,1] = PR[90,1] + 17.071;
   1:  PR[91,2] = PR[90,2] + 29.227;
   1:  PR[91,3] = PR[90,3] + 101.288;
   1:L PR[91] R[100]mm/sec CNT100;
   1:  PR[91,1] = PR[90,1] + 9.994;
   1:  PR[91,2] = PR[90,2] + 28.850;
   1:  PR[91,3] = PR[90,3] + 101.301;
   1:L PR[91] R[100]mm/sec CNT100;
   1:  PR[91,1] = PR[90,1] + 3.810;
   1:  PR[91,2] = PR[90,2] + 28.009;
   1:  PR[91,3] = PR[90,3] + 101.334;
   1:L PR[91] R[100]mm/sec CNT100;
   1:  PR[91,1] = PR[90,1] + 1.801;
   1:  PR[91,2] = PR[90,2] + 27.789;
   1:  PR[91,3] = PR[90,3] + 101.363;
   1:L PR[91] R[100]mm/sec CNT100;
   1:  PR[91,1] = PR[90,1] + -7.978;
   1:  PR[91,2] = PR[90,2] + 26.003;
   1:  PR[91,3] = PR[90,3] + 101.373;
   1:L PR[91] R[100]mm/sec CNT100;
   1:  PR[91,1] = PR[90,1] + -10.714;
   1:  PR[91,2] = PR[90,2] + 25.292;
   1:  PR[91,3] = PR[90,3] + 101.420;
   1:L PR[91] R[100]mm/sec CNT100;
   1:  PR[91,1] = PR[90,1] + -16.860;
   1:  PR[91,2] = PR[90,2] + 23.665;
   1:  PR[91,3] = PR[90,3] + 101.433;
   1:L PR[91] R[100]mm/sec CNT100;
   1:  PR[91,1] = PR[90,1] + -24.726;
   1:  PR[91,2] = PR[90,2] + 20.852;
   1:  PR[91,3] = PR[90,3] + 101.463;
   1:L PR[91] R[100]mm/sec CNT100;
   1:  PR[91,1] = PR[90,1] + -31.465;
   1:  PR[91,2] = PR[90,2] + 17.656;
   1:  PR[91,3] = PR[90,3] + 101.503;
   1:L PR[91] R[100]mm/sec CNT100;
   1:  PR[91,1] = PR[90,1] + -36.596;
   1:  PR[91,2] = PR[90,2] + 14.418;
   1:  PR[91,3] = PR[90,3] + 101.538;
   1:L PR[91] R[100]mm/sec CNT100;
   1:  PR[91,1] = PR[90,1] + -36.985;
   1:  PR[91,2] = PR[90,2] + 14.170;
   1:  PR[91,3] = PR[90,3] + 101.566;
   1:L PR[91] R[100]mm/sec CNT100;
   1:  PR[91,1] = PR[90,1] + -40.036;
   1:  PR[91,2] = PR[90,2] + 11.538;
   1:  PR[91,3] = PR[90,3] + 101.568;
   1:L PR[91] R[100]mm/sec CNT100;
   1:  PR[91,1] = PR[90,1] + -41.182;
   1:  PR[91,2] = PR[90,2] + 10.429;
   1:  PR[91,3] = PR[90,3] + 101.587;
   1:L PR[91] R[100]mm/sec CNT100;
   1:  PR[91] = PR[90];
   1:  PR[91,1] = PR[90,1] + -41.762;
   1:  PR[91,2] = PR[90,2] + 7.058;
   1:  PR[91,3] = PR[90,3] + 102.895;
   1:L PR[91] R[100]mm/sec CNT100;
   1:  PR[91,1] = PR[90,1] + -42.026;
   1:  PR[91,2] = PR[90,2] + 6.587;
   1:  PR[91,3] = PR[90,3] + 101.606;
   1:L PR[91] R[100]mm/sec CNT100;
   1:  PR[91,1] = PR[90,1] + -43.397;
   1:  PR[91,2] = PR[90,2] + 3.360;
   1:  PR[91,3] = PR[90,3] + 101.608;
   1:L PR[91] R[100]mm/sec CNT100;
   1:  PR[91,1] = PR[90,1] + -43.625;
   1:  PR[91,2] = PR[90,2] + 2.121;
   1:  PR[91,3] = PR[90,3] + 101.625;
   1:L PR[91] R[100]mm/sec CNT100;
   1:  PR[91,1] = PR[90,1] + -44.011;
   1:  PR[91,2] = PR[90,2] + -0.655;
   1:  PR[91,3] = PR[90,3] + 101.631;
   1:L PR[91] R[100]mm/sec CNT100;
   1:  PR[91,1] = PR[90,1] + -43.762;
   1:  PR[91,2] = PR[90,2] + -1.816;
   1:  PR[91,3] = PR[90,3] + 101.644;
   1:L PR[91] R[100]mm/sec CNT100;
   1:  PR[91,1] = PR[90,1] + -43.354;
   1:  PR[91,2] = PR[90,2] + -4.835;
   1:  PR[91,3] = PR[90,3] + 101.650;
   1:L PR[91] R[100]mm/sec CNT100;
   1:  PR[91,1] = PR[90,1] + -41.983;
   1:  PR[91,2] = PR[90,2] + -8.100;
   1:  PR[91,3] = PR[90,3] + 101.664;
   1:L PR[91] R[100]mm/sec CNT100;
   1:  PR[91,1] = PR[90,1] + -41.761;
   1:  PR[91,2] = PR[90,2] + -8.498;
   1:  PR[91,3] = PR[90,3] + 101.681;
   1:L PR[91] R[100]mm/sec CNT100;
   1:  PR[91,1] = PR[90,1] + -40.439;
   1:  PR[91,2] = PR[90,2] + -10.332;
   1:  PR[91,3] = PR[90,3] + 101.683;
   1:L PR[91] R[100]mm/sec CNT100;
   1:  PR[91,1] = PR[90,1] + -39.085;
   1:  PR[91,2] = PR[90,2] + -12.040;
   1:  PR[91,3] = PR[90,3] + 101.694;
   1:L PR[91] R[100]mm/sec CNT100;
   1:  PR[91,1] = PR[90,1] + -39.044;
   1:  PR[91,2] = PR[90,2] + -12.076;
   1:  PR[91,3] = PR[90,3] + 101.705;
   1:L PR[91] R[100]mm/sec CNT100;
   1:  PR[91,1] = PR[90,1] + -34.789;
   1:  PR[91,2] = PR[90,2] + -15.746;
   1:L PR[91] R[100]mm/sec CNT100;
   1:  PR[91,1] = PR[90,1] + -29.226;
   1:  PR[91,2] = PR[90,2] + -19.263;
   1:  PR[91,3] = PR[90,3] + 101.732;
   1:L PR[91] R[100]mm/sec CNT100;
   1:  PR[91,1] = PR[90,1] + -22.441;
   1:  PR[91,2] = PR[90,2] + -22.483;
   1:  PR[91,3] = PR[90,3] + 101.763;
   1:L PR[91] R[100]mm/sec CNT100;
   1:  PR[91,1] = PR[90,1] + -14.522;
   1:  PR[91,2] = PR[90,2] + -25.319;
   1:  PR[91,3] = PR[90,3] + 101.799;
   1:L PR[91] R[100]mm/sec CNT100;
   1:  PR[91,1] = PR[90,1] + -5.574;
   1:  PR[91,2] = PR[90,2] + -27.678;
   1:  PR[91,3] = PR[90,3] + 101.839;
   1:L PR[91] R[100]mm/sec CNT100;
   1:  PR[91,1] = PR[90,1] + 3.318;
   1:  PR[91,2] = PR[90,2] + -29.304;
   1:  PR[91,3] = PR[90,3] + 101.883;
   1:L PR[91] R[100]mm/sec CNT100;
   1:  PR[91,1] = PR[90,1] + 3.961;
   1:  PR[91,2] = PR[90,2] + -29.449;
   1:  PR[91,3] = PR[90,3] + 101.926;
   1:L PR[91] R[100]mm/sec CNT100;
   1:  PR[91,1] = PR[90,1] + 5.231;
   1:  PR[91,2] = PR[90,2] + -29.640;
   1:  PR[91,3] = PR[90,3] + 101.929;
   1:L PR[91] R[100]mm/sec CNT100;
   1:  PR[91,1] = PR[90,1] + 11.669;
   1:  PR[91,2] = PR[90,2] + -30.517;
   1:  PR[91,3] = PR[90,3] + 101.935;
   1:L PR[91] R[100]mm/sec CNT100;
   1:  PR[91,1] = PR[90,1] + 16.200;
   1:  PR[91,2] = PR[90,2] + -30.758;
   1:  PR[91,3] = PR[90,3] + 101.966;
   1:L PR[91] R[100]mm/sec CNT100;
   1:  PR[91,1] = PR[90,1] + 21.247;
   1:  PR[91,2] = PR[90,2] + -31.088;
   1:  PR[91,3] = PR[90,3] + 101.987;
   1:L PR[91] R[100]mm/sec CNT100;
   1:  PR[91,1] = PR[90,1] + 21.711;
   1:  PR[91,2] = PR[90,2] + -31.096;
   1:  PR[91,3] = PR[90,3] + 102.011;
   1:L PR[91] R[100]mm/sec CNT100;
   1:  PR[91,1] = PR[90,1] + 27.454;
   1:  PR[91,2] = PR[90,2] + -30.791;
   1:  PR[91,3] = PR[90,3] + 102.014;
   1:L PR[91] R[100]mm/sec CNT100;
   1:  PR[91,1] = PR[90,1] + 27.282;
   1:  PR[91,2] = PR[90,2] + -31.403;
   1:  PR[91,3] = PR[90,3] + 102.041;
   1:L PR[91] R[100]mm/sec CNT100;
   1:  PR[91,1] = PR[90,1] + 27.911;
   1:  PR[91,2] = PR[90,2] + -31.505;
   1:  PR[91,3] = PR[90,3] + 102.044;
   1:L PR[91] R[100]mm/sec CNT100;
   1:  PR[91,1] = PR[90,1] + 28.439;
   1:  PR[91,2] = PR[90,2] + -31.566;
   1:  PR[91,3] = PR[90,3] + 102.047;
   1:L PR[91] R[100]mm/sec CNT100;
   1:  PR[91,1] = PR[90,1] + 30.355;
   1:  PR[91,2] = PR[90,2] + -31.693;
   1:  PR[91,3] = PR[90,3] + 102.050;
   1:L PR[91] R[100]mm/sec CNT100;
   1:  PR[91,1] = PR[90,1] + 33.991;
   1:  PR[91,2] = PR[90,2] + -31.618;
   1:  PR[91,3] = PR[90,3] + 102.059;
   1:L PR[91] R[100]mm/sec CNT100;
   1:  PR[91,1] = PR[90,1] + 35.961;
   1:  PR[91,2] = PR[90,2] + -31.416;
   1:  PR[91,3] = PR[90,3] + 102.076;
   1:L PR[91] R[100]mm/sec CNT100;
   1:  PR[91,1] = PR[90,1] + 39.430;
   1:  PR[91,2] = PR[90,2] + -30.690;
   1:  PR[91,3] = PR[90,3] + 102.085;
   1:L PR[91] R[100]mm/sec CNT100;
   1:  PR[91,1] = PR[90,1] + 41.418;
   1:  PR[91,2] = PR[90,2] + -30.135;
   1:  PR[91,3] = PR[90,3] + 102.102;
   1:L PR[91] R[100]mm/sec CNT100;
   1:  PR[91,1] = PR[90,1] + 44.584;
   1:  PR[91,2] = PR[90,2] + -28.830;
   1:  PR[91,3] = PR[90,3] + 102.112;
   1:L PR[91] R[100]mm/sec CNT100;
   1:  PR[91,1] = PR[90,1] + 46.547;
   1:  PR[91,2] = PR[90,2] + -27.900;
   1:  PR[91,3] = PR[90,3] + 102.128;
   1:L PR[91] R[100]mm/sec CNT100;
   1:  PR[91,1] = PR[90,1] + 49.293;
   1:  PR[91,2] = PR[90,2] + -26.117;
   1:  PR[91,3] = PR[90,3] + 102.139;
   1:L PR[91] R[100]mm/sec CNT100;
   1:  PR[91,1] = PR[90,1] + 51.187;
   1:  PR[91,2] = PR[90,2] + -24.788;
   1:  PR[91,3] = PR[90,3] + 102.154;
   1:L PR[91] R[100]mm/sec CNT100;
   1:  PR[91,1] = PR[90,1] + 53.422;
   1:  PR[91,2] = PR[90,2] + -22.669;
   1:  PR[91,3] = PR[90,3] + 102.165;
   1:L PR[91] R[100]mm/sec CNT100;
   1:  PR[91,1] = PR[90,1] + 55.187;
   1:  PR[91,2] = PR[90,2] + -20.915;
   1:  PR[91,3] = PR[90,3] + 102.180;
   1:L PR[91] R[100]mm/sec CNT100;
   1:  PR[91,1] = PR[90,1] + 56.859;
   1:  PR[91,2] = PR[90,2] + -18.617;
   1:  PR[91,3] = PR[90,3] + 102.192;
   1:L PR[91] R[100]mm/sec CNT100;
   1:  PR[91,1] = PR[90,1] + 58.424;
   1:  PR[91,2] = PR[90,2] + -16.414;
   1:  PR[91,3] = PR[90,3] + 102.205;
   1:L PR[91] R[100]mm/sec CNT100;
   1:  PR[91,1] = PR[90,1] + 60.806;
   1:  PR[91,2] = PR[90,2] + -11.438;
   1:  PR[91,3] = PR[90,3] + 102.218;
   1:L PR[91] R[100]mm/sec CNT100;
   1:  PR[91,1] = PR[90,1] + 62.257;
   1:  PR[91,2] = PR[90,2] + -6.156;
   1:  PR[91,3] = PR[90,3] + 102.244;
   1:L PR[91] R[100]mm/sec CNT100;
   1:  PR[91,1] = PR[90,1] + 62.750;
   1:  PR[91,2] = PR[90,2] + -0.729;
   1:  PR[91,3] = PR[90,3] + 102.271;
   1:L PR[91] R[100]mm/sec CNT100;
   1:  PR[91,1] = PR[90,1] + 62.257;
   1:  PR[91,2] = PR[90,2] + 4.698;
   1:  PR[91,3] = PR[90,3] + 102.296;
   1:L PR[91] R[100]mm/sec CNT100;
   1:  PR[91,1] = PR[90,1] + 60.805;
   1:  PR[91,2] = PR[90,2] + 9.981;
   1:  PR[91,3] = PR[90,3] + 102.322;
   1:L PR[91] R[100]mm/sec CNT100;
   1:  PR[91,1] = PR[90,1] + 58.423;
   1:  PR[91,2] = PR[90,2] + 14.957;
   1:  PR[91,3] = PR[90,3] + 102.348;
   1:L PR[91] R[100]mm/sec CNT100;
   1:  PR[91,1] = PR[90,1] + 56.858;
   1:  PR[91,2] = PR[90,2] + 17.160;
   1:  PR[91,3] = PR[90,3] + 102.375;
   1:L PR[91] R[100]mm/sec CNT100;
   1:  PR[91,1] = PR[90,1] + 55.186;
   1:  PR[91,2] = PR[90,2] + 19.458;
   1:  PR[91,3] = PR[90,3] + 102.388;
   1:L PR[91] R[100]mm/sec CNT100;
   1:  PR[91,1] = PR[90,1] + 53.420;
   1:  PR[91,2] = PR[90,2] + 21.211;
   1:  PR[91,3] = PR[90,3] + 102.401;
   1:L PR[91] R[100]mm/sec CNT100;
   1:  PR[91,1] = PR[90,1] + 51.185;
   1:  PR[91,2] = PR[90,2] + 23.331;
   1:  PR[91,3] = PR[90,3] + 102.413;
   1:L PR[91] R[100]mm/sec CNT100;
   1:  PR[91,1] = PR[90,1] + 49.292;
   1:  PR[91,2] = PR[90,2] + 24.658;
   1:  PR[91,3] = PR[90,3] + 102.428;
   1:L PR[91] R[100]mm/sec CNT100;
   1:  PR[91,1] = PR[90,1] + 46.545;
   1:  PR[91,2] = PR[90,2] + 26.442;
   1:  PR[91,3] = PR[90,3] + 102.439;
   1:L PR[91] R[100]mm/sec CNT100;
   1:  PR[91,1] = PR[90,1] + 44.583;
   1:  PR[91,2] = PR[90,2] + 27.370;
   1:  PR[91,3] = PR[90,3] + 102.454;
   1:L PR[91] R[100]mm/sec CNT100;
   1:  PR[91,1] = PR[90,1] + 41.417;
   1:  PR[91,2] = PR[90,2] + 28.677;
   1:  PR[91,3] = PR[90,3] + 102.464;
   1:L PR[91] R[100]mm/sec CNT100;
   1:  PR[91,1] = PR[90,1] + 39.430;
   1:  PR[91,2] = PR[90,2] + 29.230;
   1:  PR[91,3] = PR[90,3] + 102.481;
   1:L PR[91] R[100]mm/sec CNT100;
   1:  PR[91,1] = PR[90,1] + 35.960;
   1:  PR[91,2] = PR[90,2] + 29.958;
   1:  PR[91,3] = PR[90,3] + 102.491;
   1:L PR[91] R[100]mm/sec CNT100;
   1:  PR[91,1] = PR[90,1] + 33.991;
   1:  PR[91,2] = PR[90,2] + 30.159;
   1:  PR[91,3] = PR[90,3] + 102.507;
   1:L PR[91] R[100]mm/sec CNT100;
   1:  PR[91,1] = PR[90,1] + 30.354;
   1:  PR[91,2] = PR[90,2] + 30.234;
   1:  PR[91,3] = PR[90,3] + 102.517;
   1:L PR[91] R[100]mm/sec CNT100;
   1:  PR[91,1] = PR[90,1] + 28.440;
   1:  PR[91,2] = PR[90,2] + 30.107;
   1:  PR[91,3] = PR[90,3] + 102.534;
   1:L PR[91] R[100]mm/sec CNT100;
   1:  PR[91,1] = PR[90,1] + 27.822;
   1:  PR[91,2] = PR[90,2] + 30.035;
   1:  PR[91,3] = PR[90,3] + 102.543;
   1:L PR[91] R[100]mm/sec CNT100;
   1:  PR[91,1] = PR[90,1] + 24.884;
   1:  PR[91,2] = PR[90,2] + 29.559;
   1:  PR[91,3] = PR[90,3] + 102.546;
   1:L PR[91] R[100]mm/sec CNT100;
   1:  PR[91,1] = PR[90,1] + 21.832;
   1:  PR[91,2] = PR[90,2] + 29.638;
   1:  PR[91,3] = PR[90,3] + 102.560;
   1:L PR[91] R[100]mm/sec CNT100;
   1:  PR[91,1] = PR[90,1] + 21.252;
   1:  PR[91,2] = PR[90,2] + 29.629;
   1:  PR[91,3] = PR[90,3] + 102.575;
   1:L PR[91] R[100]mm/sec CNT100;
   1:  PR[91,1] = PR[90,1] + 16.200;
   1:  PR[91,2] = PR[90,2] + 29.300;
   1:  PR[91,3] = PR[90,3] + 102.578;
   1:L PR[91] R[100]mm/sec CNT100;
   1:  PR[91,1] = PR[90,1] + 11.670;
   1:  PR[91,2] = PR[90,2] + 29.058;
   1:  PR[91,3] = PR[90,3] + 102.602;
   1:L PR[91] R[100]mm/sec CNT100;
   1:  PR[91,1] = PR[90,1] + 5.231;
   1:  PR[91,2] = PR[90,2] + 28.182;
   1:  PR[91,3] = PR[90,3] + 102.623;
   1:L PR[91] R[100]mm/sec CNT100;
   1:  PR[91,1] = PR[90,1] + 3.961;
   1:  PR[91,2] = PR[90,2] + 27.990;
   1:  PR[91,3] = PR[90,3] + 102.654;
   1:L PR[91] R[100]mm/sec CNT100;
   1:  PR[91,1] = PR[90,1] + 3.318;
   1:  PR[91,2] = PR[90,2] + 27.846;
   1:  PR[91,3] = PR[90,3] + 102.660;
   1:L PR[91] R[100]mm/sec CNT100;
   1:  PR[91,1] = PR[90,1] + -5.574;
   1:  PR[91,2] = PR[90,2] + 26.220;
   1:  PR[91,3] = PR[90,3] + 102.664;
   1:L PR[91] R[100]mm/sec CNT100;
   1:  PR[91,1] = PR[90,1] + -14.522;
   1:  PR[91,2] = PR[90,2] + 23.860;
   1:  PR[91,3] = PR[90,3] + 102.707;
   1:L PR[91] R[100]mm/sec CNT100;
   1:  PR[91,1] = PR[90,1] + -22.442;
   1:  PR[91,2] = PR[90,2] + 21.024;
   1:  PR[91,3] = PR[90,3] + 102.751;
   1:L PR[91] R[100]mm/sec CNT100;
   1:  PR[91,1] = PR[90,1] + -27.000;
   1:  PR[91,2] = PR[90,2] + 18.869;
   1:  PR[91,3] = PR[90,3] + 102.791;
   1:L PR[91] R[100]mm/sec CNT100;
   1:  PR[91,1] = PR[90,1] + -29.223;
   1:  PR[91,2] = PR[90,2] + 17.806;
   1:  PR[91,3] = PR[90,3] + 102.815;
   1:L PR[91] R[100]mm/sec CNT100;
   1:  PR[91,1] = PR[90,1] + -34.789;
   1:  PR[91,2] = PR[90,2] + 14.288;
   1:  PR[91,3] = PR[90,3] + 102.826;
   1:L PR[91] R[100]mm/sec CNT100;
   1:  PR[91,1] = PR[90,1] + -39.088;
   1:  PR[91,2] = PR[90,2] + 10.578;
   1:  PR[91,3] = PR[90,3] + 102.858;
   1:L PR[91] R[100]mm/sec CNT100;
   1:  PR[91,1] = PR[90,1] + -40.442;
   1:  PR[91,2] = PR[90,2] + 8.868;
   1:  PR[91,3] = PR[90,3] + 102.885;
   1:L PR[91] R[100]mm/sec CNT100;
   1:  PR[91] = PR[90];
   1:  PR[91,1] = PR[90,1] + -40.854;
   1:  PR[91,2] = PR[90,2] + 4.880;
   1:  PR[91,3] = PR[90,3] + 104.195;
   1:L PR[91] R[100]mm/sec CNT100;
   1:  PR[91,1] = PR[90,1] + -41.599;
   1:  PR[91,2] = PR[90,2] + 3.126;
   1:  PR[91,3] = PR[90,3] + 102.905;
   1:L PR[91] R[100]mm/sec CNT100;
   1:  PR[91,1] = PR[90,1] + -41.622;
   1:  PR[91,2] = PR[90,2] + 3.002;
   1:  PR[91,3] = PR[90,3] + 102.915;
   1:L PR[91] R[100]mm/sec CNT100;
   1:  PR[91,1] = PR[90,1] + -42.130;
   1:  PR[91,2] = PR[90,2] + -0.655;
   1:L PR[91] R[100]mm/sec CNT100;
   1:  PR[91,1] = PR[90,1] + -42.075;
   1:  PR[91,2] = PR[90,2] + -0.913;
   1:  PR[91,3] = PR[90,3] + 102.933;
   1:L PR[91] R[100]mm/sec CNT100;
   1:  PR[91,1] = PR[90,1] + -41.574;
   1:  PR[91,2] = PR[90,2] + -4.626;
   1:  PR[91,3] = PR[90,3] + 102.934;
   1:L PR[91] R[100]mm/sec CNT100;
   1:  PR[91,1] = PR[90,1] + -40.853;
   1:  PR[91,2] = PR[90,2] + -6.342;
   1:  PR[91,3] = PR[90,3] + 102.952;
   1:L PR[91] R[100]mm/sec CNT100;
   1:  PR[91,1] = PR[90,1] + -39.945;
   1:  PR[91,2] = PR[90,2] + -8.308;
   1:  PR[91,3] = PR[90,3] + 102.961;
   1:L PR[91] R[100]mm/sec CNT100;
   1:  PR[91,1] = PR[90,1] + -36.918;
   1:  PR[91,2] = PR[90,2] + -12.128;
   1:  PR[91,3] = PR[90,3] + 102.972;
   1:L PR[91] R[100]mm/sec CNT100;
   1:  PR[91,1] = PR[90,1] + -32.589;
   1:  PR[91,2] = PR[90,2] + -15.867;
   1:  PR[91,3] = PR[90,3] + 102.995;
   1:L PR[91] R[100]mm/sec CNT100;
   1:  PR[91,1] = PR[90,1] + -26.988;
   1:  PR[91,2] = PR[90,2] + -19.410;
   1:  PR[91,3] = PR[90,3] + 103.022;
   1:L PR[91] R[100]mm/sec CNT100;
   1:  PR[91,1] = PR[90,1] + -20.156;
   1:  PR[91,2] = PR[90,2] + -22.656;
   1:  PR[91,3] = PR[90,3] + 103.054;
   1:L PR[91] R[100]mm/sec CNT100;
   1:  PR[91,1] = PR[90,1] + -12.183;
   1:  PR[91,2] = PR[90,2] + -25.515;
   1:  PR[91,3] = PR[90,3] + 103.091;
   1:L PR[91] R[100]mm/sec CNT100;
   1:  PR[91,1] = PR[90,1] + -3.172;
   1:  PR[91,2] = PR[90,2] + -27.894;
   1:  PR[91,3] = PR[90,3] + 103.131;
   1:L PR[91] R[100]mm/sec CNT100;
   1:  PR[91,1] = PR[90,1] + 2.669;
   1:  PR[91,2] = PR[90,2] + -28.962;
   1:  PR[91,3] = PR[90,3] + 103.176;
   1:L PR[91] R[100]mm/sec CNT100;
   1:  PR[91,1] = PR[90,1] + 5.288;
   1:  PR[91,2] = PR[90,2] + -29.551;
   1:  PR[91,3] = PR[90,3] + 103.204;
   1:L PR[91] R[100]mm/sec CNT100;
   1:  PR[91,1] = PR[90,1] + 10.524;
   1:  PR[91,2] = PR[90,2] + -30.341;
   1:  PR[91,3] = PR[90,3] + 103.217;
   1:L PR[91] R[100]mm/sec CNT100;
   1:  PR[91,1] = PR[90,1] + 13.345;
   1:  PR[91,2] = PR[90,2] + -30.725;
   1:  PR[91,3] = PR[90,3] + 103.243;
   1:L PR[91] R[100]mm/sec CNT100;
   1:  PR[91,1] = PR[90,1] + 15.328;
   1:  PR[91,2] = PR[90,2] + -30.830;
   1:  PR[91,3] = PR[90,3] + 103.256;
   1:L PR[91] R[100]mm/sec CNT100;
   1:  PR[91,1] = PR[90,1] + 22.782;
   1:  PR[91,2] = PR[90,2] + -31.317;
   1:  PR[91,3] = PR[90,3] + 103.266;
   1:L PR[91] R[100]mm/sec CNT100;
   1:  PR[91,1] = PR[90,1] + 23.522;
   1:  PR[91,2] = PR[90,2] + -31.330;
   1:  PR[91,3] = PR[90,3] + 103.302;
   1:L PR[91] R[100]mm/sec CNT100;
   1:  PR[91,1] = PR[90,1] + 28.057;
   1:  PR[91,2] = PR[90,2] + -31.089;
   1:  PR[91,3] = PR[90,3] + 103.305;
   1:L PR[91] R[100]mm/sec CNT100;
   1:  PR[91,1] = PR[90,1] + 27.901;
   1:  PR[91,2] = PR[90,2] + -31.644;
   1:  PR[91,3] = PR[90,3] + 103.327;
   1:L PR[91] R[100]mm/sec CNT100;
   1:  PR[91,1] = PR[90,1] + 28.182;
   1:  PR[91,2] = PR[90,2] + -31.677;
   1:  PR[91,3] = PR[90,3] + 103.330;
   1:L PR[91] R[100]mm/sec CNT100;
   1:  PR[91,1] = PR[90,1] + 31.039;
   1:  PR[91,2] = PR[90,2] + -31.866;
   1:  PR[91,3] = PR[90,3] + 103.331;
   1:L PR[91] R[100]mm/sec CNT100;
   1:  PR[91,1] = PR[90,1] + 33.625;
   1:  PR[91,2] = PR[90,2] + -31.813;
   1:  PR[91,3] = PR[90,3] + 103.345;
   1:L PR[91] R[100]mm/sec CNT100;
   1:  PR[91,1] = PR[90,1] + 36.676;
   1:  PR[91,2] = PR[90,2] + -31.499;
   1:  PR[91,3] = PR[90,3] + 103.358;
   1:L PR[91] R[100]mm/sec CNT100;
   1:  PR[91,1] = PR[90,1] + 38.974;
   1:  PR[91,2] = PR[90,2] + -31.019;
   1:  PR[91,3] = PR[90,3] + 103.372;
   1:L PR[91] R[100]mm/sec CNT100;
   1:  PR[91,1] = PR[90,1] + 42.154;
   1:  PR[91,2] = PR[90,2] + -30.132;
   1:  PR[91,3] = PR[90,3] + 103.384;
   1:L PR[91] R[100]mm/sec CNT100;
   1:  PR[91,1] = PR[90,1] + 44.040;
   1:  PR[91,2] = PR[90,2] + -29.354;
   1:  PR[91,3] = PR[90,3] + 103.399;
   1:L PR[91] R[100]mm/sec CNT100;
   1:  PR[91,1] = PR[90,1] + 47.292;
   1:  PR[91,2] = PR[90,2] + -27.813;
   1:  PR[91,3] = PR[90,3] + 103.409;
   1:L PR[91] R[100]mm/sec CNT100;
   1:  PR[91,1] = PR[90,1] + 48.678;
   1:  PR[91,2] = PR[90,2] + -26.913;
   1:  PR[91,3] = PR[90,3] + 103.426;
   1:L PR[91] R[100]mm/sec CNT100;
   1:  PR[91,1] = PR[90,1] + 51.932;
   1:  PR[91,2] = PR[90,2] + -24.631;
   1:  PR[91,3] = PR[90,3] + 103.434;
   1:L PR[91] R[100]mm/sec CNT100;
   1:  PR[91,1] = PR[90,1] + 52.776;
   1:  PR[91,2] = PR[90,2] + -23.830;
   1:  PR[91,3] = PR[90,3] + 103.454;
   1:L PR[91] R[100]mm/sec CNT100;
   1:  PR[91,1] = PR[90,1] + 55.913;
   1:  PR[91,2] = PR[90,2] + -20.714;
   1:  PR[91,3] = PR[90,3] + 103.459;
   1:L PR[91] R[100]mm/sec CNT100;
   1:  PR[91,1] = PR[90,1] + 59.142;
   1:  PR[91,2] = PR[90,2] + -16.184;
   1:  PR[91,3] = PR[90,3] + 103.480;
   1:L PR[91] R[100]mm/sec CNT100;
   1:  PR[91,1] = PR[90,1] + 61.491;
   1:  PR[91,2] = PR[90,2] + -11.347;
   1:  PR[91,3] = PR[90,3] + 103.507;
   1:L PR[91] R[100]mm/sec CNT100;
   1:  PR[91,1] = PR[90,1] + 61.672;
   1:  PR[91,2] = PR[90,2] + -10.773;
   1:  PR[91,3] = PR[90,3] + 103.533;
   1:L PR[91] R[100]mm/sec CNT100;
   1:  PR[91,1] = PR[90,1] + 62.960;
   1:  PR[91,2] = PR[90,2] + -6.180;
   1:  PR[91,3] = PR[90,3] + 103.536;
   1:L PR[91] R[100]mm/sec CNT100;
   1:  PR[91,1] = PR[90,1] + 63.465;
   1:  PR[91,2] = PR[90,2] + -0.726;
   1:  PR[91,3] = PR[90,3] + 103.559;
   1:L PR[91] R[100]mm/sec CNT100;
   1:  PR[91,1] = PR[90,1] + 63.094;
   1:  PR[91,2] = PR[90,2] + 3.412;
   1:  PR[91,3] = PR[90,3] + 103.585;
   1:L PR[91] R[100]mm/sec CNT100;
   1:  PR[91,1] = PR[90,1] + 62.962;
   1:  PR[91,2] = PR[90,2] + 4.714;
   1:  PR[91,3] = PR[90,3] + 103.605;
   1:L PR[91] R[100]mm/sec CNT100;
   1:  PR[91,1] = PR[90,1] + 61.670;
   1:  PR[91,2] = PR[90,2] + 9.319;
   1:  PR[91,3] = PR[90,3] + 103.611;
   1:L PR[91] R[100]mm/sec CNT100;
   1:  PR[91,1] = PR[90,1] + 61.489;
   1:  PR[91,2] = PR[90,2] + 9.892;
   1:  PR[91,3] = PR[90,3] + 103.634;
   1:L PR[91] R[100]mm/sec CNT100;
   1:  PR[91,1] = PR[90,1] + 59.138;
   1:  PR[91,2] = PR[90,2] + 14.731;
   1:  PR[91,3] = PR[90,3] + 103.637;
   1:L PR[91] R[100]mm/sec CNT100;
   1:  PR[91,1] = PR[90,1] + 55.908;
   1:  PR[91,2] = PR[90,2] + 19.261;
   1:  PR[91,3] = PR[90,3] + 103.663;
   1:L PR[91] R[100]mm/sec CNT100;
   1:  PR[91,1] = PR[90,1] + 52.770;
   1:  PR[91,2] = PR[90,2] + 22.376;
   1:  PR[91,3] = PR[90,3] + 103.690;
   1:L PR[91] R[100]mm/sec CNT100;
   1:  PR[91,1] = PR[90,1] + 51.925;
   1:  PR[91,2] = PR[90,2] + 23.177;
   1:  PR[91,3] = PR[90,3] + 103.711;
   1:L PR[91] R[100]mm/sec CNT100;
   1:  PR[91,1] = PR[90,1] + 48.672;
   1:  PR[91,2] = PR[90,2] + 25.458;
   1:  PR[91,3] = PR[90,3] + 103.716;
   1:L PR[91] R[100]mm/sec CNT100;
   1:  PR[91,1] = PR[90,1] + 47.285;
   1:  PR[91,2] = PR[90,2] + 26.358;
   1:  PR[91,3] = PR[90,3] + 103.736;
   1:L PR[91] R[100]mm/sec CNT100;
   1:  PR[91,1] = PR[90,1] + 44.034;
   1:  PR[91,2] = PR[90,2] + 27.897;
   1:  PR[91,3] = PR[90,3] + 103.743;
   1:L PR[91] R[100]mm/sec CNT100;
   1:  PR[91,1] = PR[90,1] + 42.147;
   1:  PR[91,2] = PR[90,2] + 28.676;
   1:  PR[91,3] = PR[90,3] + 103.761;
   1:L PR[91] R[100]mm/sec CNT100;
   1:  PR[91,1] = PR[90,1] + 38.968;
   1:  PR[91,2] = PR[90,2] + 29.560;
   1:  PR[91,3] = PR[90,3] + 103.771;
   1:L PR[91] R[100]mm/sec CNT100;
   1:  PR[91,1] = PR[90,1] + 36.669;
   1:  PR[91,2] = PR[90,2] + 30.042;
   1:  PR[91,3] = PR[90,3] + 103.786;
   1:L PR[91] R[100]mm/sec CNT100;
   1:  PR[91,1] = PR[90,1] + 33.620;
   1:  PR[91,2] = PR[90,2] + 30.354;
   1:  PR[91,3] = PR[90,3] + 103.798;
   1:L PR[91] R[100]mm/sec CNT100;
   1:  PR[91,1] = PR[90,1] + 31.032;
   1:  PR[91,2] = PR[90,2] + 30.407;
   1:  PR[91,3] = PR[90,3] + 103.812;
   1:L PR[91] R[100]mm/sec CNT100;
   1:  PR[91,1] = PR[90,1] + 28.177;
   1:  PR[91,2] = PR[90,2] + 30.217;
   1:  PR[91,3] = PR[90,3] + 103.825;
   1:L PR[91] R[100]mm/sec CNT100;
   1:  PR[91,1] = PR[90,1] + 27.233;
   1:  PR[91,2] = PR[90,2] + 30.107;
   1:  PR[91,3] = PR[90,3] + 103.839;
   1:L PR[91] R[100]mm/sec CNT100;
   1:  PR[91,1] = PR[90,1] + 25.494;
   1:  PR[91,2] = PR[90,2] + 29.826;
   1:  PR[91,3] = PR[90,3] + 103.843;
   1:L PR[91] R[100]mm/sec CNT100;
   1:  PR[91,1] = PR[90,1] + 23.688;
   1:  PR[91,2] = PR[90,2] + 29.873;
   1:  PR[91,3] = PR[90,3] + 103.852;
   1:L PR[91] R[100]mm/sec CNT100;
   1:  PR[91,1] = PR[90,1] + 22.790;
   1:  PR[91,2] = PR[90,2] + 29.858;
   1:  PR[91,3] = PR[90,3] + 103.860;
   1:L PR[91] R[100]mm/sec CNT100;
   1:  PR[91,1] = PR[90,1] + 15.328;
   1:  PR[91,2] = PR[90,2] + 29.372;
   1:  PR[91,3] = PR[90,3] + 103.865;
   1:L PR[91] R[100]mm/sec CNT100;
   1:  PR[91,1] = PR[90,1] + 13.346;
   1:  PR[91,2] = PR[90,2] + 29.266;
   1:  PR[91,3] = PR[90,3] + 103.900;
   1:L PR[91] R[100]mm/sec CNT100;
   1:  PR[91,1] = PR[90,1] + 10.526;
   1:  PR[91,2] = PR[90,2] + 28.882;
   1:  PR[91,3] = PR[90,3] + 103.910;
   1:L PR[91] R[100]mm/sec CNT100;
   1:  PR[91,1] = PR[90,1] + 5.288;
   1:  PR[91,2] = PR[90,2] + 28.093;
   1:  PR[91,3] = PR[90,3] + 103.924;
   1:L PR[91] R[100]mm/sec CNT100;
   1:  PR[91,1] = PR[90,1] + 2.669;
   1:  PR[91,2] = PR[90,2] + 27.503;
   1:  PR[91,3] = PR[90,3] + 103.949;
   1:L PR[91] R[100]mm/sec CNT100;
   1:  PR[91,1] = PR[90,1] + -3.172;
   1:  PR[91,2] = PR[90,2] + 26.435;
   1:  PR[91,3] = PR[90,3] + 103.962;
   1:L PR[91] R[100]mm/sec CNT100;
   1:  PR[91,1] = PR[90,1] + -12.183;
   1:  PR[91,2] = PR[90,2] + 24.056;
   1:  PR[91,3] = PR[90,3] + 103.991;
   1:L PR[91] R[100]mm/sec CNT100;
   1:  PR[91,1] = PR[90,1] + -20.156;
   1:  PR[91,2] = PR[90,2] + 21.198;
   1:  PR[91,3] = PR[90,3] + 104.035;
   1:L PR[91] R[100]mm/sec CNT100;
   1:  PR[91,1] = PR[90,1] + -26.988;
   1:  PR[91,2] = PR[90,2] + 17.952;
   1:  PR[91,3] = PR[90,3] + 104.076;
   1:L PR[91] R[100]mm/sec CNT100;
   1:  PR[91,1] = PR[90,1] + -32.589;
   1:  PR[91,2] = PR[90,2] + 14.408;
   1:  PR[91,3] = PR[90,3] + 104.112;
   1:L PR[91] R[100]mm/sec CNT100;
   1:  PR[91,1] = PR[90,1] + -36.918;
   1:  PR[91,2] = PR[90,2] + 10.669;
   1:  PR[91,3] = PR[90,3] + 104.144;
   1:L PR[91] R[100]mm/sec CNT100;
   1:  PR[91,1] = PR[90,1] + -39.945;
   1:  PR[91,2] = PR[90,2] + 6.849;
   1:  PR[91,3] = PR[90,3] + 104.172;
   1:L PR[91] R[100]mm/sec CNT100;
   1:  PR[91] = PR[90];
   1:  PR[91,1] = PR[90,1] + -39.573;
   1:  PR[91,2] = PR[90,2] + 3.064;
   1:  PR[91,3] = PR[90,3] + 105.495;
   1:L PR[91] R[100]mm/sec CNT100;
   1:  PR[91,1] = PR[90,1] + -40.152;
   1:  PR[91,2] = PR[90,2] + -0.729;
   1:  PR[91,3] = PR[90,3] + 104.216;
   1:L PR[91] R[100]mm/sec CNT100;
   1:  PR[91,1] = PR[90,1] + -39.573;
   1:  PR[91,2] = PR[90,2] + -4.523;
   1:  PR[91,3] = PR[90,3] + 104.234;
   1:L PR[91] R[100]mm/sec CNT100;
   1:  PR[91,1] = PR[90,1] + -37.797;
   1:  PR[91,2] = PR[90,2] + -8.370;
   1:  PR[91,3] = PR[90,3] + 104.253;
   1:L PR[91] R[100]mm/sec CNT100;
   1:  PR[91,1] = PR[90,1] + -34.746;
   1:  PR[91,2] = PR[90,2] + -12.223;
   1:  PR[91,3] = PR[90,3] + 104.273;
   1:L PR[91] R[100]mm/sec CNT100;
   1:  PR[91,1] = PR[90,1] + -34.005;
   1:  PR[91,2] = PR[90,2] + -12.868;
   1:  PR[91,3] = PR[90,3] + 104.297;
   1:L PR[91] R[100]mm/sec CNT100;
   1:  PR[91,1] = PR[90,1] + -30.390;
   1:  PR[91,2] = PR[90,2] + -15.987;
   1:  PR[91,3] = PR[90,3] + 104.302;
   1:L PR[91] R[100]mm/sec CNT100;
   1:  PR[91,1] = PR[90,1] + -24.750;
   1:  PR[91,2] = PR[90,2] + -19.558;
   1:  PR[91,3] = PR[90,3] + 104.325;
   1:L PR[91] R[100]mm/sec CNT100;
   1:  PR[91,1] = PR[90,1] + -17.871;
   1:  PR[91,2] = PR[90,2] + -22.829;
   1:  PR[91,3] = PR[90,3] + 104.357;
   1:L PR[91] R[100]mm/sec CNT100;
   1:  PR[91,1] = PR[90,1] + -9.843;
   1:  PR[91,2] = PR[90,2] + -25.710;
   1:  PR[91,3] = PR[90,3] + 104.394;
   1:L PR[91] R[100]mm/sec CNT100;
   1:  PR[91,1] = PR[90,1] + -0.771;
   1:  PR[91,2] = PR[90,2] + -28.110;
   1:  PR[91,3] = PR[90,3] + 104.436;
   1:L PR[91] R[100]mm/sec CNT100;
   1:  PR[91,1] = PR[90,1] + 2.021;
   1:  PR[91,2] = PR[90,2] + -28.620;
   1:  PR[91,3] = PR[90,3] + 104.481;
   1:L PR[91] R[100]mm/sec CNT100;
   1:  PR[91,1] = PR[90,1] + 6.614;
   1:  PR[91,2] = PR[90,2] + -29.654;
   1:  PR[91,3] = PR[90,3] + 104.495;
   1:L PR[91] R[100]mm/sec CNT100;
   1:  PR[91,1] = PR[90,1] + 14.674;
   1:  PR[91,2] = PR[90,2] + -30.869;
   1:  PR[91,3] = PR[90,3] + 104.518;
   1:L PR[91] R[100]mm/sec CNT100;
   1:  PR[91,1] = PR[90,1] + 15.053;
   1:  PR[91,2] = PR[90,2] + -30.940;
   1:  PR[91,3] = PR[90,3] + 104.557;
   1:L PR[91] R[100]mm/sec CNT100;
   1:  PR[91,1] = PR[90,1] + 24.318;
   1:  PR[91,2] = PR[90,2] + -31.546;
   1:  PR[91,3] = PR[90,3] + 104.559;
   1:L PR[91] R[100]mm/sec CNT100;
   1:  PR[91,1] = PR[90,1] + 25.334;
   1:  PR[91,2] = PR[90,2] + -31.564;
   1:  PR[91,3] = PR[90,3] + 104.604;
   1:L PR[91] R[100]mm/sec CNT100;
   1:  PR[91,1] = PR[90,1] + 28.659;
   1:  PR[91,2] = PR[90,2] + -31.388;
   1:  PR[91,3] = PR[90,3] + 104.609;
   1:L PR[91] R[100]mm/sec CNT100;
   1:  PR[91,1] = PR[90,1] + 28.535;
   1:  PR[91,2] = PR[90,2] + -31.828;
   1:  PR[91,3] = PR[90,3] + 104.625;
